ABB RobotStudio station: COMPAS_RRC_IRB-4600-40_2.55_ws_zhaw_hslu.rspag

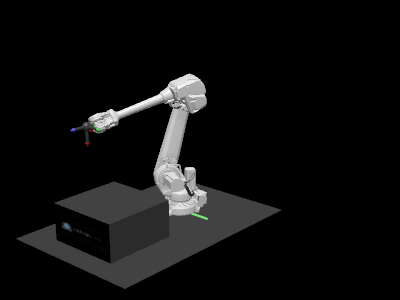
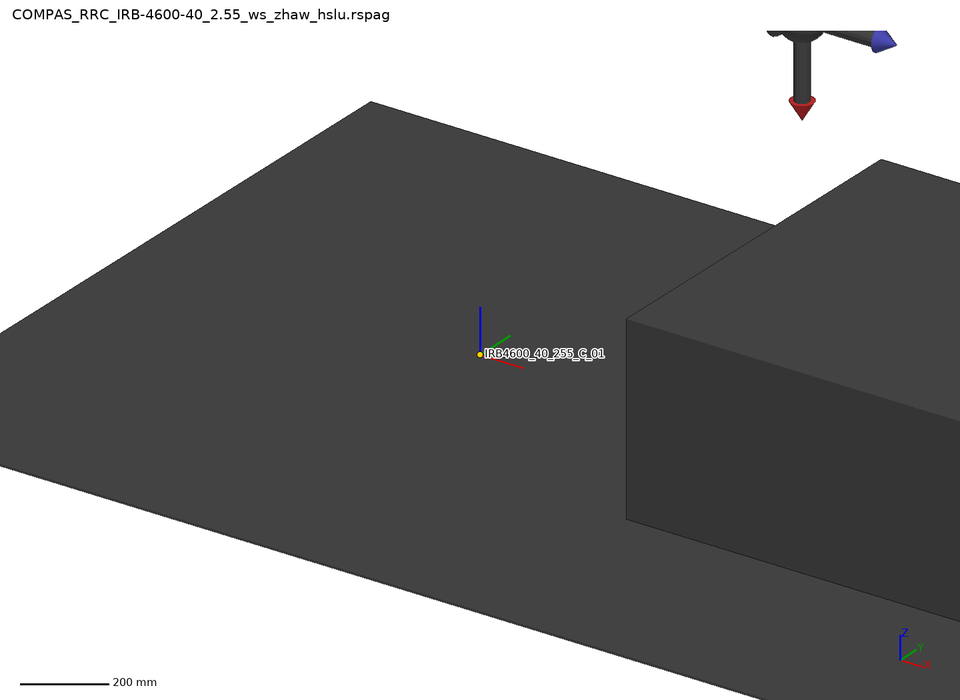
[picture v1: parts stored in the station drawn from their meshes, with robot base, taught points and paths (robot models come from the ABB library and are not in the file)]
--- station ---
Station COMPAS_RRC_IRB-4600-40_2.55 (saved by RobotStudio 22.2.10013.1)
Controller vIRB4600-40-2.55-RW11
  mechanical unit ROB_1: IRB4600_40_255_C_01, 6 joints, base frame (0, 0, 0) mm
Layout (positions relative to the parent item):
  - IRB4600_40_255_C_01 [mechanism] at (0, 0, 0) mm; joint values [-0.4275, -0.3109, 0.5805, -1.0418, -0.501, 0.9829] (rad or m)
      links: Base, Link1, Link2, Link3, Link4, Link5, Link6
  - Tool [graphiccomponentgroup] at (1145.78, -460.56, 1367.89) mm, rotated rx -105.47 ry 90 rz -105.47 deg
    - Tool X [part], size 50 x 60 x 60 mm
    - Tool Y [part], size 60 x 50 x 60 mm
    - Tool Z [part], size 60 x 60 x 50 mm
    - Base [part] at (1428.26, 0, 1185.08) mm, rotated rx 180 ry 0 rz -180 deg, size 272.5 x 272.4 x 270 mm
    - Tool X TubeTrace [smart component]
        properties: TraceObject=(none); ActiveTube=(none); Mechanism=IRB4600_40_255_C_01; Flange=Tool0; Parent=(none); Flange Offset=[0.26 0 0.06]; Tube Diameter=0.03; Color (RGB)=[255 255 255]; Color=-65536; Min Distance=0.001; Redraw Rate (ms)=10; NoOfBodies=278; Remove Geometry=true; Transient=false
        signals: DI Execute, DI NewTrace, DI Clear, DO TraceCreated
    - Tool Y TubeTrace [smart component]
        properties: TraceObject=(none); ActiveTube=(none); Mechanism=IRB4600_40_255_C_01; Flange=Tool0; Parent=(none); Flange Offset=[0 0.26 0.06]; Tube Diameter=0.03; Color (RGB)=[255 255 255]; Color=-16711872; Min Distance=0.001; Redraw Rate (ms)=10; NoOfBodies=278; Remove Geometry=true; Transient=false
        signals: DI Execute, DI NewTrace, DI Clear, DO TraceCreated
    - Tool Z TubeTrace [smart component]
        properties: TraceObject=(none); ActiveTube=(none); Mechanism=IRB4600_40_255_C_01; Flange=Tool0; Parent=(none); Flange Offset=[0 0 0.32]; Tube Diameter=0.03; Color (RGB)=[255 255 255]; Color=-16776961; Min Distance=0.001; Redraw Rate (ms)=10; NoOfBodies=278; Remove Geometry=true; Transient=false
        signals: DI Execute, DI NewTrace, DI Clear, DO TraceCreated
  - Example_Setup [graphiccomponentgroup]
    - Ground [part], size 3000 x 2000 x 5 mm
    - Table [part], size 1000 x 1000 x 500 mm
Attachment: Tool is attached to IRB4600_40_255_C_01 / Link6
Station logic (signal -> signal, property => property):
  vIRB4600-40-2.55-RW11.do_X -> Tool X TubeTrace.Execute
  vIRB4600-40-2.55-RW11.do_Y -> Tool Y TubeTrace.Execute
  vIRB4600-40-2.55-RW11.do_Z -> Tool Z TubeTrace.Execute

--- Backups/vIRB4600-40-2.55-RW11/RAPID/TASK1/PROGMOD/RRC_Example.mod ---
MODULE RRC_Example
    !***********************************************************************************
    !
    ! ETH Zurich / Robotic Fabrication Lab
    ! HIB C 13 / Stefano-Franscini-Platz 1
    ! CH-8093 Zurich
    !
    !***********************************************************************************
    !
    ! PROJECT     :  RRC - Rapid Robot Communication
    !
    ! FUNCTION    :  Example modul for the project
    !
    ! AUTHOR      :  Philippe Fleischmann
    !
    ! EMAIL       :  rrc@arch.ethz.ch
    !
    ! HISTORY     :  2019.02.22
    !
    ! Copyright   :  ETH Zurich (CH) 2019
    !                - Philippe Fleischmann
    !                - Michael Lyrenmann
    !                - Gonzalo Casas
    !
    ! License     :  This code base is governed by an EULA (End-User License Agreement)
    !                which you have received together with the software.
    !                You are not allowed to use the software on a real robots
    !                without a signed EULA.
    !
    !                A copy of the EULA content is in the controller task (T_CTRL).
    !
    !***********************************************************************************

    !************************************************
    ! Declaration :     tooldata
    !************************************************
    !
    TASK PERS tooldata t_RRC_Tool_X:=[TRUE,[[260,0,60],[0.707106781,0,0.707106781,0]],[15,[0,0,60],[1,0,0,0],0,0,0]];
    TASK PERS tooldata t_RRC_Tool_Y:=[TRUE,[[0,260,60],[0.707106781,-0.707106781,0,0]],[15,[0,0,60],[1,0,0,0],0,0,0]];
    TASK PERS tooldata t_RRC_Tool_Z:=[TRUE,[[0,0,320],[1,0,0,0]],[15,[0,0,60],[1,0,0,0],0,0,0]];

    !************************************************
    ! Declaration :     wobjdata
    !************************************************
    !
    TASK PERS wobjdata ob_RRC_Workplace:=[FALSE,TRUE,"",[[750,-500,500],[1,0,0,0]],[[0,0,0],[1,0,0,0]]];

ENDMODULE

--- Backups/vIRB4600-40-2.55-RW11/RAPID/TASK1/PROGMOD/RRC_Main.mod ---
MODULE RRC_Main
    !***********************************************************************************
    !
    ! ETH Zurich / Robotic Fabrication Lab
    ! HIB C 13 / Stefano-Franscini-Platz 1
    ! CH-8093 Zurich
    !
    !***********************************************************************************
    !
    ! PROJECT     :  RRC - Rapid Robot Communication
    !
    ! FUNCTION    :  Main modul for the project
    !
    ! AUTHOR      :  Philippe Fleischmann
    !
    ! EMAIL       :  rrc@arch.ethz.ch
    !
    ! HISTORY     :  2019.02.22
    !
    ! Copyright   :  ETH Zurich (CH) 2019
    !                - Philippe Fleischmann
    !                - Michael Lyrenmann
    !                - Gonzalo Casas
    !
    ! License     :  This code base is governed by an EULA (End-User License Agreement)
    !                which you have received together with the software.
    !                You are not allowed to use the software on a real robots
    !                without a signed EULA.
    !
    !                A copy of the EULA content is in the controller task (T_CTRL).
    !
    !***********************************************************************************

    !************************************************
    ! Function    :     main
    ! Programmer  :     Philippe Fleischmann
    ! Date        :     2019.02.22
    !***************** ETH Zurich *******************
    !
    PROC main()
        !****************************!
        !                            !
        !   #####   #####    ####    !
        !   #    #  #    #  #    #   !
        !   #    #  #    #  #        !
        !   #####   #####   #        !
        !   #   #   #   #   #    #   !
        !   #    #  #    #   ####    !
        !                            !
        !****************************!
        !
        r_RRC_Main;
    ENDPROC

ENDMODULE

--- Backups/vIRB4600-40-2.55-RW11/RAPID/TASK1/SYSMOD/RRC_Base_DataTask_Rob.sys ---
MODULE RRC_Base_DataTask_Rob (SYSMODULE)
    !***********************************************************************************
    !
    ! ETH Zurich / Robotic Fabrication Lab
    ! HIB C 13 / Stefano-Franscini-Platz 1
    ! CH-8093 Zurich
    !
    !***********************************************************************************
    !
    ! PROJECT     :  RRC - Rapid Robot Communication
    !
    ! FUNCTION    :  Base Data Task Library
    !
    ! AUTHOR      :  Philippe Fleischmann
    !
    ! EMAIL       :  rrc@arch.ethz.ch
    !
    ! HISTORY     :  2019.02.22
    !
    ! Copyright   :  ETH Zurich (CH) 2019
    !                - Philippe Fleischmann
    !                - Michael Lyrenmann
    !                - Gonzalo Casas
    !
    ! License     :  This code base is governed by an EULA (End-User License Agreement)
    !                which you have received together with the software.
    !                You are not allowed to use the software on a real robots
    !                without a signed EULA.
    !
    !                A copy of the EULA content is in the controller task (T_CTRL).
    !
    !***********************************************************************************

    !************************************************
    ! Declaration :     num
    !************************************************
    !
    TASK PERS num n_RRC_Answer:=0;
    TASK PERS num n_RRC_Act_S_ID:=4;
    TASK PERS num n_RRC_Time:=1;
    TASK PERS num n_RRC_Acc:=100;
    TASK PERS num n_RRC_Ramp:=100;
    TASK PERS num n_RRC_Override:=100;
    TASK PERS num n_RRC_MaxTCP:=500;
    TASK PERS num n_RRC_FloatValue:=42;

    !************************************************
    ! Declaration :     string
    !************************************************
    !
    TASK PERS string st_RRC_UIAnswer:="Set my Speed";
    TASK PERS string st_RRC_ActMsg1:="Requested speed is not posible, minimal value is 0.1 mm/s";
    TASK PERS string st_RRC_ActMsg2:="Submited speed : 0.0 mm/s";
    TASK PERS string st_RRC_ActMsg3:="";
    TASK PERS string st_RRC_ActMsg4:="";
    TASK PERS string st_RRC_ActMsg5:="";
    TASK PERS string st_RRC_ActBtn1:="50 mm/s";
    TASK PERS string st_RRC_ActBtn2:="100 mm/s";
    TASK PERS string st_RRC_ActBtn3:="Set my Speed";
    TASK PERS string st_RRC_ActBtn4:="";
    TASK PERS string st_RRC_ActBtn5:="";
    TASK PERS string st_RRC_Header:="Update Speed";
    TASK PERS string st_RRC_TPWrite:="Moving to position on target_frame";
    TASK PERS string st_RRC_StringValue:="Custom Text";

    !************************************************
    ! Declaration :     tooldata
    !************************************************
    !
    TASK PERS tooldata t_RRC_Act:=[TRUE,[[0,0,320],[1,0,0,0]],[15,[0,0,60],[1,0,0,0],0,0,0]];

    !************************************************
    ! Declaration :     wobjdata
    !************************************************
    !
    TASK PERS wobjdata ob_RRC_Act:=[FALSE,TRUE,"",[[750,-500,500],[1,0,0,0]],[[0,0,0],[1,0,0,0]]];

    !************************************************
    ! Declaration :     speeddata
    !************************************************
    !
    CONST speeddata v_RRC_Default:=[25,500,5000,1000];
    TASK PERS speeddata v_RRC_Act:=[200,500,5000,1000];

    !************************************************
    ! Declaration :     zonedata
    !************************************************
    !
    TASK PERS zonedata z_RRC_Act:=[TRUE,0,0,0,0,0,0];

    !************************************************
    ! Declaration :     jointtarget
    !************************************************
    !
    TASK PERS jointtarget jp_RRC_Act:=[[-24.4963,-17.8131,33.2614,-59.6898,-28.7042,56.3166],[9E+9,9E+9,9E+9,9E+9,9E+9,9E+9]];

    !************************************************
    ! Declaration :     robtarget
    !************************************************
    !
    TASK PERS robtarget p_RRC_Act:=[[715.775,39.4411,867.894],[0.707107,0,0.707107,0],[0,0,-1,0],[9E+9,9E+9,9E+9,9E+9,9E+9,9E+9]];

    !************************************************
    ! Declaration :     signaldo
    !************************************************
    !
    VAR signaldo do_RRC_Act;

    !************************************************
    ! Declaration :     signalgo
    !************************************************
    !
    VAR signalgo go_RRC_Act;

    !************************************************
    ! Declaration :     signalao
    !************************************************
    !
    VAR signalao ao_RRC_Act;

    !************************************************
    ! Declaration :     signaldi
    !************************************************
    !
    VAR signaldi di_RRC_Act;

    !************************************************
    ! Declaration :     signalgi
    !************************************************
    !
    VAR signalgi gi_RRC_Act;

    !************************************************
    ! Declaration :     signalai
    !************************************************
    !
    VAR signalai ai_RRC_Act;

    !************************************************
    ! Declaration :     signalai
    !************************************************
    !
    VAR clock ck_RRC_StopWatch;

ENDMODULE

--- Backups/vIRB4600-40-2.55-RW11/RAPID/TASK1/SYSMOD/RRC_Base_Feedback_Rob.sys ---
MODULE RRC_Base_Feedback_Rob(SYSMODULE)
    !***********************************************************************************
    !
    ! ETH Zurich / Robotic Fabrication Lab
    ! HIB C 13 / Stefano-Franscini-Platz 1
    ! CH-8093 Zurich
    !
    !***********************************************************************************
    !
    ! PROJECT     :  RRC - Rapid Robot Communication
    !
    ! FUNCTION    :  Base Feedback Library
    !
    ! AUTHOR      :  Philippe Fleischmann
    !
    ! EMAIL       :  rrc@arch.ethz.ch
    !
    ! HISTORY     :  2019.02.22
    !
    ! Copyright   :  ETH Zurich (CH) 2019
    !                - Philippe Fleischmann
    !                - Michael Lyrenmann
    !                - Gonzalo Casas
    !
    ! License     :  This code base is governed by an EULA (End-User License Agreement)
    !                which you have received together with the software.
    !                You are not allowed to use the software on a real robots
    !                without a signed EULA.
    !
    !                A copy of the EULA content is in the controller task (T_CTRL).
    !
    !***********************************************************************************

    !************************************************
    ! Function    :     Feedback add string
    ! Programmer  :     Philippe Fleischmann
    ! Date        :     2019.02.22
    !***************** ETH Zurich *******************
    !
    PROC r_RRC_FAddString(string stString)
        !
        ! Increase feedback string counter
        Incr n_RRC_CounterFStr;
        !
        ! Select string to add
        TEST n_RRC_CounterFStr
        CASE 1:
            !
            ! Add string
            bm_RRC_ActSenMsgRob.Data.St1:=stString;
        CASE 2:
            !
            ! Add string
            bm_RRC_ActSenMsgRob.Data.St2:=stString;
        CASE 3:
            !
            ! Add string
            bm_RRC_ActSenMsgRob.Data.St3:=stString;
        CASE 4:
            !
            ! Add string
            bm_RRC_ActSenMsgRob.Data.St4:=stString;
        CASE 5:
            !
            ! Add string
            bm_RRC_ActSenMsgRob.Data.St5:=stString;
        DEFAULT:
            !
            ! Program error
            r_RRC_ProgError;
        ENDTEST
        !
        ! Update string counter
        bm_RRC_ActSenMsgRob.Data.St_Cnt:=n_RRC_CounterFStr;
        RETURN ;
    ERROR
        ! Placeholder for Error Code...
    ENDPROC

    !************************************************
    ! Function    :     Feedback add value
    ! Programmer  :     Philippe Fleischmann
    ! Date        :     2019.02.22
    !***************** ETH Zurich *******************
    !
    PROC r_RRC_FAddValue(num nValue)
        !
        ! Increase feedback value counter
        Incr n_RRC_CounterFVal;
        !
        ! Select value to add
        TEST n_RRC_CounterFVal
        CASE 1:
            !
            ! Add value
            bm_RRC_ActSenMsgRob.Data.V1:=nValue;
        CASE 2:
            !
            ! Add value
            bm_RRC_ActSenMsgRob.Data.V2:=nValue;
        CASE 3:
            !
            ! Add value
            bm_RRC_ActSenMsgRob.Data.V3:=nValue;
        CASE 4:
            !
            ! Add value
            bm_RRC_ActSenMsgRob.Data.V4:=nValue;
        CASE 5:
            !
            ! Add value
            bm_RRC_ActSenMsgRob.Data.V5:=nValue;
        CASE 6:
            !
            ! Add value
            bm_RRC_ActSenMsgRob.Data.V6:=nValue;
        CASE 7:
            !
            ! Add value
            bm_RRC_ActSenMsgRob.Data.V7:=nValue;
        CASE 8:
            !
            ! Add value
            bm_RRC_ActSenMsgRob.Data.V8:=nValue;
        CASE 9:
            !
            ! Add value
            bm_RRC_ActSenMsgRob.Data.V9:=nValue;
        CASE 10:
            !
            ! Add value
            bm_RRC_ActSenMsgRob.Data.V10:=nValue;
        CASE 11:
            !
            ! Add value
            bm_RRC_ActSenMsgRob.Data.V11:=nValue;
        CASE 12:
            !
            ! Add value
            bm_RRC_ActSenMsgRob.Data.V12:=nValue;
        CASE 13:
            !
            ! Add value
            bm_RRC_ActSenMsgRob.Data.V13:=nValue;
        CASE 14:
            !
            ! Add value
            bm_RRC_ActSenMsgRob.Data.V14:=nValue;
        CASE 15:
            !
            ! Add value
            bm_RRC_ActSenMsgRob.Data.V15:=nValue;
        CASE 16:
            !
            ! Add value
            bm_RRC_ActSenMsgRob.Data.V16:=nValue;
        CASE 17:
            !
            ! Add value
            bm_RRC_ActSenMsgRob.Data.V17:=nValue;
        CASE 18:
            !
            ! Add value
            bm_RRC_ActSenMsgRob.Data.V18:=nValue;
        CASE 19:
            !
            ! Add value
            bm_RRC_ActSenMsgRob.Data.V19:=nValue;
        CASE 20:
            !
            ! Add value
            bm_RRC_ActSenMsgRob.Data.V20:=nValue;
        CASE 21:
            !
            ! Add value
            bm_RRC_ActSenMsgRob.Data.V21:=nValue;
        CASE 22:
            !
            ! Add value
            bm_RRC_ActSenMsgRob.Data.V22:=nValue;
        CASE 23:
            !
            ! Add value
            bm_RRC_ActSenMsgRob.Data.V23:=nValue;
        CASE 24:
            !
            ! Add value
            bm_RRC_ActSenMsgRob.Data.V24:=nValue;
        CASE 25:
            !
            ! Add value
            bm_RRC_ActSenMsgRob.Data.V25:=nValue;
        CASE 26:
            !
            ! Add value
            bm_RRC_ActSenMsgRob.Data.V26:=nValue;
        CASE 27:
            !
            ! Add value
            bm_RRC_ActSenMsgRob.Data.V27:=nValue;
        CASE 28:
            !
            ! Add value
            bm_RRC_ActSenMsgRob.Data.V28:=nValue;
        CASE 29:
            !
            ! Add value
            bm_RRC_ActSenMsgRob.Data.V29:=nValue;
        CASE 30:
            !
            ! Add value
            bm_RRC_ActSenMsgRob.Data.V30:=nValue;
        DEFAULT:
            !
            ! Program error
            r_RRC_ProgError;
        ENDTEST
        !
        ! Update value counter
        bm_RRC_ActSenMsgRob.Data.V_Cnt:=n_RRC_CounterFVal;
        RETURN ;
    ERROR
        ! Placeholder for Error Code...
    ENDPROC

    !************************************************
    ! Function    :     Feedback done
    ! Programmer  :     Philippe Fleischmann
    ! Date        :     2019.02.22
    !***************** ETH Zurich *******************
    !
    PROC r_RRC_FDone()
        !
        ! Add Sqz_ID from Client in Feedback ID
        bm_RRC_ActSenMsgRob.Data.F_ID:=bm_RRC_RecBufferRob{n_RRC_ChaNr,n_RRC_ReadPtrRecBuf}.Data.S_ID;
        !
        ! Instruction
        bm_RRC_ActSenMsgRob.Data.Instr:=bm_RRC_RecBufferRob{n_RRC_ChaNr,n_RRC_ReadPtrRecBuf}.Data.Instr;
        !
        ! Feedback
        bm_RRC_ActSenMsgRob.Data.Feedb:="Done";
        RETURN ;
    ERROR
        ! Placeholder for Error Code...
    ENDPROC

    !************************************************
    ! Function    :     Feedback Position
    ! Programmer  :     Philippe Fleischmann
    ! Date        :     2019.02.22
    !***************** ETH Zurich *******************
    !
    PROC r_RRC_FPos(num nFL)
        !
        ! Check feedback level
        TEST nFL
        CASE 10001:
            !
            ! add robot position after robot is in position
            r_RRC_FActRobT;
        CASE 10002:
            !
            ! add fly by robot positon
            r_RRC_FActRobT\FlyBy;
        CASE 10003:
            !
            ! add robot joints after robot is in position
            r_RRC_FActJointT;
        CASE 10004:
            !
            ! add fly by joints positon
            r_RRC_FActJointT\FlyBy;
        ENDTEST
        RETURN ;
    ERROR
        ! Placeholder for Error Code...
    ENDPROC

    !************************************************
    ! Function    :     Feedback actual jointtarget
    ! Programmer  :     Philippe Fleischmann
    ! Date        :     2019.02.22
    !***************** ETH Zurich *******************
    !
    PROC r_RRC_FActJointT(\switch FlyBy)
        !
        ! Read actual jointtartet
        r_RRC_ReadActJointT\FlyBy?FlyBy;
        !
        ! Read robot axis
        r_RRC_FAddValue jp_RRC_Act.robax.rax_1;
        r_RRC_FAddValue jp_RRC_Act.robax.rax_2;
        r_RRC_FAddValue jp_RRC_Act.robax.rax_3;
        r_RRC_FAddValue jp_RRC_Act.robax.rax_4;
        r_RRC_FAddValue jp_RRC_Act.robax.rax_5;
        r_RRC_FAddValue jp_RRC_Act.robax.rax_6;
        !
        ! Read external axis
        r_RRC_FAddValue jp_RRC_Act.extax.eax_a;
        r_RRC_FAddValue jp_RRC_Act.extax.eax_b;
        r_RRC_FAddValue jp_RRC_Act.extax.eax_c;
        !
        ! Reserve for unused external axis
        r_RRC_FAddValue jp_RRC_Act.extax.eax_d;
        r_RRC_FAddValue jp_RRC_Act.extax.eax_e;
        r_RRC_FAddValue jp_RRC_Act.extax.eax_f;
        RETURN ;
    ERROR
        ! Placeholder for Error Code...
    ENDPROC

    !************************************************
    ! Function    :     Feedback actual robtarget
    ! Programmer  :     Philippe Fleischmann
    ! Date        :     2019.02.22
    !***************** ETH Zurich *******************
    !
    PROC r_RRC_FActRobT(\switch FlyBy)
        !
        ! Read actual robtarget
        r_RRC_ReadActRobT\FlyBy?FlyBy;
        !
        ! Read actual translation
        r_RRC_FAddValue p_RRC_Act.trans.x;
        r_RRC_FAddValue p_RRC_Act.trans.y;
        r_RRC_FAddValue p_RRC_Act.trans.z;
        !
        ! Read actual rotation (Quaternions)
        r_RRC_FAddValue p_RRC_Act.rot.q1;
        r_RRC_FAddValue p_RRC_Act.rot.q2;
        r_RRC_FAddValue p_RRC_Act.rot.q3;
        r_RRC_FAddValue p_RRC_Act.rot.q4;
        !
        ! Read actual external axis
        r_RRC_FAddValue p_RRC_Act.extax.eax_a;
        r_RRC_FAddValue p_RRC_Act.extax.eax_b;
        r_RRC_FAddValue p_RRC_Act.extax.eax_c;
        !
        ! Reserve for unused external axis
        r_RRC_FAddValue p_RRC_Act.extax.eax_d;
        r_RRC_FAddValue p_RRC_Act.extax.eax_e;
        r_RRC_FAddValue p_RRC_Act.extax.eax_f;
        RETURN ;
    ERROR
        ! Placeholder for Error Code...
    ENDPROC

    !************************************************
    ! Function    :     Feedback error
    ! Programmer  :     Philippe Fleischmann
    ! Date        :     2019.02.22
    !***************** ETH Zurich *******************
    !
    PROC r_RRC_FError()
        !
        ! Feedback error with feedback code
        bm_RRC_ActSenMsgRob.Data.Feedb:="Done FError "+NumToStr(bm_RRC_RecBufferRob{n_RRC_ChaNr,n_RRC_ReadPtrRecBuf}.Data.F_Lev,0);
        RETURN ;
    ERROR
        ! Placeholder for Error Code...
    ENDPROC
ENDMODULE

--- Backups/vIRB4600-40-2.55-RW11/RAPID/TASK1/SYSMOD/RRC_Base_Instructions_Rob.sys ---
MODULE RRC_Base_Instructions_Rob(SYSMODULE)
    !***********************************************************************************
    !
    ! ETH Zurich / Robotic Fabrication Lab
    ! HIB C 13 / Stefano-Franscini-Platz 1
    ! CH-8093 Zurich
    !
    !***********************************************************************************
    !
    ! PROJECT     :  RRC - Rapid Robot Communication
    !
    ! FUNCTION    :  Base Instracion Library
    !
    ! AUTHOR      :  Philippe Fleischmann
    !
    ! EMAIL       :  rrc@arch.ethz.ch
    !
    ! HISTORY     :  2019.02.22
    !
    ! Copyright   :  ETH Zurich (CH) 2019
    !                - Philippe Fleischmann
    !                - Michael Lyrenmann
    !                - Gonzalo Casas
    !
    ! License     :  This code base is governed by an EULA (End-User License Agreement)
    !                which you have received together with the software.
    !                You are not allowed to use the software on a real robots
    !                without a signed EULA.
    !
    !                A copy of the EULA content is in the controller task (T_CTRL).
    !
    !***********************************************************************************

    !************************************************
    ! Function    :     Move to Joints (MoveAbsJ)
    ! Programmer  :     Philippe Fleischmann
    ! Date        :     2019.02.22
    !***************** ETH Zurich *******************
    !
    PROC r_RRC_MoveToJoints()
        !
        ! Read and set jonttarget
        r_RRC_RasJointtarget;
        !
        ! Read and set tcp speed
        r_RRC_RasTCPSpeed bm_RRC_RecBufferRob{n_RRC_ChaNr,n_RRC_ReadPtrRecBuf}.Data.V13;
        !
        ! Read and set zone
        r_RRC_RasZone bm_RRC_RecBufferRob{n_RRC_ChaNr,n_RRC_ReadPtrRecBuf}.Data.V14;
        !
        ! Move robot
        MoveAbsJ jp_RRC_Act,v_RRC_Act,z_RRC_Act,t_RRC_Act;
        !
        ! Feedback
        IF bm_RRC_RecBufferRob{n_RRC_ChaNr,n_RRC_ReadPtrRecBuf}.Data.F_Lev>0 THEN
            !
            ! Instruction done
            r_RRC_FDone;
            !
            ! Check additional feedback
            IF bm_RRC_RecBufferRob{n_RRC_ChaNr,n_RRC_ReadPtrRecBuf}.Data.F_Lev>1 THEN
                !
                ! Cenerate feedback
                TEST bm_RRC_RecBufferRob{n_RRC_ChaNr,n_RRC_ReadPtrRecBuf}.Data.F_Lev
                DEFAULT:
                    !
                    ! Not defined
                    !
                    ! Feedback not supported
                    r_RRC_FError;
                ENDTEST
            ENDIF
            !
            ! Move message in send buffer
            r_RRC_MovMsgToSenBufRob n_RRC_ChaNr;
        ENDIF
        RETURN ;
    ERROR
        ! Placeholder for Error Code...
    ENDPROC

    !************************************************
    ! Function    :     Move to (MoveL or MoveJ)
    ! Programmer  :     Philippe Fleischmann
    ! Date        :     2019.02.22
    !***************** ETH Zurich *******************
    !
    PROC r_RRC_MoveTo()
        !
        ! Read and set robtarget
        r_RRC_RASRobtarget\stMoveType:=bm_RRC_RecBufferRob{n_RRC_ChaNr,n_RRC_ReadPtrRecBuf}.Data.st1;
        !
        ! Read and set tcp speed
        r_RRC_RasTCPSpeed bm_RRC_RecBufferRob{n_RRC_ChaNr,n_RRC_ReadPtrRecBuf}.Data.V14;
        !
        ! Read and set zone
        r_RRC_RasZone bm_RRC_RecBufferRob{n_RRC_ChaNr,n_RRC_ReadPtrRecBuf}.Data.V15;
        !
        ! Select move type
        IF bm_RRC_RecBufferRob{n_RRC_ChaNr,n_RRC_ReadPtrRecBuf}.Data.st1="L" OR bm_RRC_RecBufferRob{n_RRC_ChaNr,n_RRC_ReadPtrRecBuf}.Data.st1="FrameL" THEN
            !
            ! Linear
            !
            !
            ! Deactivate configuration check
            ConfL\Off;
            !
            ! Move robot
            MoveL p_RRC_Act,v_RRC_Act,z_RRC_Act,t_RRC_Act\WObj:=ob_RRC_Act;
            !
            ! Activate configuration check
            ConfL\On;
        ELSE
            !
            ! Joint
            !
            !
            ! Deactivate configuration check
            ConfJ\Off;
            !
            ! Move robot
            MoveJ p_RRC_Act,v_RRC_Act,z_RRC_Act,t_RRC_Act\WObj:=ob_RRC_Act;
            !
            ! Activate configuration check
            ConfJ\On;
        ENDIF
        !
        ! Feedback
        IF bm_RRC_RecBufferRob{n_RRC_ChaNr,n_RRC_ReadPtrRecBuf}.Data.F_Lev>0 THEN
            !
            ! Instruction done
            r_RRC_FDone;
            !
            ! Check additional feedback
            IF bm_RRC_RecBufferRob{n_RRC_ChaNr,n_RRC_ReadPtrRecBuf}.Data.F_Lev>1 THEN
                !
                ! Cenerate feedback
                TEST bm_RRC_RecBufferRob{n_RRC_ChaNr,n_RRC_ReadPtrRecBuf}.Data.F_Lev
                DEFAULT:
                    !
                    ! Not defined
                    !
                    ! Feedback not supported
                    r_RRC_FError;
                ENDTEST
            ENDIF
            !
            ! Move message in send buffer
            r_RRC_MovMsgToSenBufRob n_RRC_ChaNr;
        ENDIF
        RETURN ;
    ERROR
        ! Placeholder for Error Code...
    ENDPROC

    !************************************************
    ! Function    :     Set analog output (SetAO)
    ! Programmer  :     Philippe Fleischmann
    ! Date        :     2019.02.22
    !***************** ETH Zurich *******************
    !
    PROC r_RRC_SetAnalog()
        !
        ! Get actual output
        GetDataVal bm_RRC_RecBufferRob{n_RRC_ChaNr,n_RRC_ReadPtrRecBuf}.Data.St1,ao_RRC_Act;
        !
        ! Set actual output
        SetAO ao_RRC_Act,bm_RRC_RecBufferRob{n_RRC_ChaNr,n_RRC_ReadPtrRecBuf}.Data.V1;
        !
        ! Feedback
        IF bm_RRC_RecBufferRob{n_RRC_ChaNr,n_RRC_ReadPtrRecBuf}.Data.F_Lev>0 THEN
            !
            ! Cenerate feedback
            TEST bm_RRC_RecBufferRob{n_RRC_ChaNr,n_RRC_ReadPtrRecBuf}.Data.F_Lev
            CASE 1:
                !
                ! Instruction done
                r_RRC_FDone;
            DEFAULT:
                !
                ! Feedback not supported
                r_RRC_FError;
            ENDTEST
            !
            ! Move message in send buffer
            r_RRC_MovMsgToSenBufRob n_RRC_ChaNr;
        ENDIF
        RETURN ;
    ERROR
        ! Placeholder for Error Code...
    ENDPROC

    !************************************************
    ! Function    :     Read ananlog input ((AInput)
    ! Programmer  :     Philippe Fleischmann
    ! Date        :     2019.02.22
    !***************** ETH Zurich *******************
    !
    PROC r_RRC_ReadAnalog()
        !
        ! Get actual output
        GetDataVal bm_RRC_RecBufferRob{n_RRC_ChaNr,n_RRC_ReadPtrRecBuf}.Data.St1,ai_RRC_Act;
        !
        ! Add standard feedback instruction done
        r_RRC_FDone;
        !
        ! Read input value and add it to feedback
        r_RRC_FAddValue AInput(ai_RRC_Act);
        !
        ! Feedback
        IF bm_RRC_RecBufferRob{n_RRC_ChaNr,n_RRC_ReadPtrRecBuf}.Data.F_Lev>1 THEN
            !
            ! Check additional feedback
            TEST bm_RRC_RecBufferRob{n_RRC_ChaNr,n_RRC_ReadPtrRecBuf}.Data.F_Lev
            CASE 10001,10002,10003,10004:
                !
                ! add robot position
                r_RRC_FPos bm_RRC_RecBufferRob{n_RRC_ChaNr,n_RRC_ReadPtrRecBuf}.Data.F_Lev;
            DEFAULT:
                !
                ! Not defined
                !
                ! Feedback not supported
                r_RRC_FError;
            ENDTEST
        ENDIF
        !
        ! Move message in send buffer
        r_RRC_MovMsgToSenBufRob n_RRC_ChaNr;
        RETURN ;
    ERROR
        ! Placeholder for Error Code...
    ENDPROC

    !************************************************
    ! Function    :     Set group output (SetGO)
    ! Programmer  :     Philippe Fleischmann
    ! Date        :     2019.02.22
    !***************** ETH Zurich *******************
    !
    PROC r_RRC_SetGroup()
        !
        ! Get actual output
        GetDataVal bm_RRC_RecBufferRob{n_RRC_ChaNr,n_RRC_ReadPtrRecBuf}.Data.St1,go_RRC_Act;
        !
        ! Set actual output
        SetGO go_RRC_Act,bm_RRC_RecBufferRob{n_RRC_ChaNr,n_RRC_ReadPtrRecBuf}.Data.V1;
        !
        ! Feedback
        IF bm_RRC_RecBufferRob{n_RRC_ChaNr,n_RRC_ReadPtrRecBuf}.Data.F_Lev>0 THEN
            !
            ! Cenerate feedback
            TEST bm_RRC_RecBufferRob{n_RRC_ChaNr,n_RRC_ReadPtrRecBuf}.Data.F_Lev
            CASE 1:
                !
                ! Instruction done
                r_RRC_FDone;
            DEFAULT:
                !
                ! Feedback not supported
                r_RRC_FError;
            ENDTEST
            !
            ! Move message in send buffer
            r_RRC_MovMsgToSenBufRob n_RRC_ChaNr;
        ENDIF
        RETURN ;
    ERROR
        ! Placeholder for Error Code...
    ENDPROC

    !************************************************
    ! Function    :     Read group input (GInput)
    ! Programmer  :     Philippe Fleischmann
    ! Date        :     2019.02.22
    !***************** ETH Zurich *******************
    !
    PROC r_RRC_ReadGroup()
        !
        ! Get actual output
        GetDataVal bm_RRC_RecBufferRob{n_RRC_ChaNr,n_RRC_ReadPtrRecBuf}.Data.St1,gi_RRC_Act;
        !
        ! Add standard feedback instruction done
        r_RRC_FDone;
        !
        ! Read input value and add it to feedback
        r_RRC_FAddValue GInput(gi_RRC_Act);
        !
        ! Feedback
        IF bm_RRC_RecBufferRob{n_RRC_ChaNr,n_RRC_ReadPtrRecBuf}.Data.F_Lev>1 THEN
            !
            ! Check additional feedback
            TEST bm_RRC_RecBufferRob{n_RRC_ChaNr,n_RRC_ReadPtrRecBuf}.Data.F_Lev
            CASE 10001,10002,10003,10004:
                !
                ! add robot position
                r_RRC_FPos bm_RRC_RecBufferRob{n_RRC_ChaNr,n_RRC_ReadPtrRecBuf}.Data.F_Lev;
            DEFAULT:
                !
                ! Not defined
                !
                ! Feedback not supported
                r_RRC_FError;
            ENDTEST
        ENDIF
        !
        ! Move message in send buffer
        r_RRC_MovMsgToSenBufRob n_RRC_ChaNr;
        RETURN ;
    ERROR
        ! Placeholder for Error Code...
    ENDPROC

    !************************************************
    ! Function    :     Set digital output (SetDO)
    ! Programmer  :     Philippe Fleischmann
    ! Date        :     2019.02.22
    !***************** ETH Zurich *******************
    !
    PROC r_RRC_SetDigital()
        !
        ! Get actual output
        GetDataVal bm_RRC_RecBufferRob{n_RRC_ChaNr,n_RRC_ReadPtrRecBuf}.Data.St1,do_RRC_Act;
        !
        ! Set actual output
        SetDO do_RRC_Act,bm_RRC_RecBufferRob{n_RRC_ChaNr,n_RRC_ReadPtrRecBuf}.Data.V1;
        !
        ! Feedback
        IF bm_RRC_RecBufferRob{n_RRC_ChaNr,n_RRC_ReadPtrRecBuf}.Data.F_Lev>0 THEN
            !
            ! Cenerate feedback
            TEST bm_RRC_RecBufferRob{n_RRC_ChaNr,n_RRC_ReadPtrRecBuf}.Data.F_Lev
            CASE 1:
                !
                ! Instruction done
                r_RRC_FDone;
            DEFAULT:
                !
                ! Feedback not supported
                r_RRC_FError;
            ENDTEST
            !
            ! Move message in send buffer
            r_RRC_MovMsgToSenBufRob n_RRC_ChaNr;
        ENDIF
        RETURN ;
    ERROR
        ! Placeholder for Error Code...
    ENDPROC

    !************************************************
    ! Function    :     Pulse digital output (PulsDo)
    ! Programmer  :     Philippe Fleischmann
    ! Date        :     2019.02.22
    !***************** ETH Zurich *******************
    !
    PROC r_RRC_PulseDigital()
        !
        ! Get actual output
        GetDataVal bm_RRC_RecBufferRob{n_RRC_ChaNr,n_RRC_ReadPtrRecBuf}.Data.St1,do_RRC_Act;
        !
        ! Set actual output
        PulseDO\High\PLength:=bm_RRC_RecBufferRob{n_RRC_ChaNr,n_RRC_ReadPtrRecBuf}.Data.V1,do_RRC_Act;
        !
        ! Feedback
        IF bm_RRC_RecBufferRob{n_RRC_ChaNr,n_RRC_ReadPtrRecBuf}.Data.F_Lev>0 THEN
            !
            ! Cenerate feedback
            TEST bm_RRC_RecBufferRob{n_RRC_ChaNr,n_RRC_ReadPtrRecBuf}.Data.F_Lev
            CASE 1:
                !
                ! Instruction done
                r_RRC_FDone;
            DEFAULT:
                !
                ! Feedback not supported
                r_RRC_FError;
            ENDTEST
            !
            ! Move message in send buffer
            r_RRC_MovMsgToSenBufRob n_RRC_ChaNr;
        ENDIF
        RETURN ;
    ERROR
        ! Placeholder for Error Code...
    ENDPROC

    !************************************************
    ! Function    :     Read digital input (DInput)
    ! Programmer  :     Philippe Fleischmann
    ! Date        :     2019.02.22
    !***************** ETH Zurich *******************
    !
    PROC r_RRC_ReadDigital()
        !
        ! Get actual output
        GetDataVal bm_RRC_RecBufferRob{n_RRC_ChaNr,n_RRC_ReadPtrRecBuf}.Data.St1,di_RRC_Act;
        !
        ! Add standard feedback instruction done
        r_RRC_FDone;
        !
        ! Read input value and add it to feedback
        r_RRC_FAddValue DInput(Di_RRC_Act);
        !
        ! Feedback
        IF bm_RRC_RecBufferRob{n_RRC_ChaNr,n_RRC_ReadPtrRecBuf}.Data.F_Lev>1 THEN
            !
            ! Check additional feedback
            TEST bm_RRC_RecBufferRob{n_RRC_ChaNr,n_RRC_ReadPtrRecBuf}.Data.F_Lev
            CASE 10001,10002,10003,10004:
                !
                ! add robot position
                r_RRC_FPos bm_RRC_RecBufferRob{n_RRC_ChaNr,n_RRC_ReadPtrRecBuf}.Data.F_Lev;
            DEFAULT:
                !
                ! Not defined
                ! Feedback not supported
                r_RRC_FError;
            ENDTEST
        ENDIF
        !
        ! Move message in send buffer
        r_RRC_MovMsgToSenBufRob n_RRC_ChaNr;
        RETURN ;
    ERROR
        ! Placeholder for Error Code...
    ENDPROC

    !************************************************
    ! Function    :     Set tool (tooldata)
    ! Programmer  :     Philippe Fleischmann
    ! Date        :     2019.02.22
    !***************** ETH Zurich *******************
    !
    PROC r_RRC_SetTool()
        VAR tooldata tX:=[TRUE,[[0,0,0],[1,0,0,0]],[0,[0,0,0],[1,0,0,0],0,0,0]];
        !
        ! Get tool
        GetDataVal bm_RRC_RecBufferRob{n_RRC_ChaNr,n_RRC_ReadPtrRecBuf}.Data.St1,tX;
        !
        ! Set t_RRC_Act
        t_RRC_Act:=tX;
        !
        ! Feedback
        IF bm_RRC_RecBufferRob{n_RRC_ChaNr,n_RRC_ReadPtrRecBuf}.Data.F_Lev>0 THEN
            !
            ! Instruction done
            r_RRC_FDone;
            !
            ! Check additional feedback
            IF bm_RRC_RecBufferRob{n_RRC_ChaNr,n_RRC_ReadPtrRecBuf}.Data.F_Lev>1 THEN
                !
                ! Cenerate feedback
                TEST bm_RRC_RecBufferRob{n_RRC_ChaNr,n_RRC_ReadPtrRecBuf}.Data.F_Lev
                CASE 10001:
                    !
                    ! Tooldata
                    ! String 1 from Client
                    r_RRC_FAddString bm_RRC_RecBufferRob{n_RRC_ChaNr,n_RRC_ReadPtrRecBuf}.Data.St1;
                    !
                    ! String 2 Structure of parameter information
                    r_RRC_FAddString "Feedback -Tool -Robhold -Pos -Orient -Mass";
                    !
                    ! String 3 roboter hold tool yes or no
                    IF t_RRC_Act.robhold=TRUE r_RRC_FAddString "Yes";
                    IF t_RRC_Act.robhold=FALSE r_RRC_FAddString "No";
                    !
                    ! Value 1..3 TCP position xyz
                    r_RRC_FAddValue t_RRC_Act.tframe.trans.x;
                    r_RRC_FAddValue t_RRC_Act.tframe.trans.y;
                    r_RRC_FAddValue t_RRC_Act.tframe.trans.z;
                    !
                    ! Value 4..7 TCP orientation q1..q4
                    r_RRC_FAddValue t_RRC_Act.tframe.rot.q1;
                    r_RRC_FAddValue t_RRC_Act.tframe.rot.q2;
                    r_RRC_FAddValue t_RRC_Act.tframe.rot.q3;
                    r_RRC_FAddValue t_RRC_Act.tframe.rot.q4;
                    !
                    ! Value 8 Tool mass
                    r_RRC_FAddValue t_RRC_Act.tload.mass;
                DEFAULT:
                    !
                    ! Feedback not supported
                    r_RRC_FError;
                ENDTEST
            ENDIF
            !
            ! Move message in send buffer
            r_RRC_MovMsgToSenBufRob n_RRC_ChaNr;
        ENDIF
        RETURN ;
    ERROR
        ! Placeholder for Error Code...
    ENDPROC

    !************************************************
    ! Function    :     Set work object (wobjdata)
    ! Programmer  :     Philippe Fleischmann
    ! Date        :     2019.02.22
    !***************** ETH Zurich *******************
    !
    PROC r_RRC_SetWorkObject()
        VAR wobjdata obX:=[FALSE,TRUE,"",[[0,0,0],[1,0,0,0]],[[0,0,0],[1,0,0,0]]];
        !
        ! Get workobject
        GetDataVal bm_RRC_RecBufferRob{n_RRC_ChaNr,n_RRC_ReadPtrRecBuf}.Data.St1,obX;
        !
        ! Set ob_RRC_Act
        ob_RRC_Act:=obX;
        !
        ! Feedback
        IF bm_RRC_RecBufferRob{n_RRC_ChaNr,n_RRC_ReadPtrRecBuf}.Data.F_Lev>0 THEN
            !
            ! Instruction done
            r_RRC_FDone;
            !
            ! Check additional feedback
            IF bm_RRC_RecBufferRob{n_RRC_ChaNr,n_RRC_ReadPtrRecBuf}.Data.F_Lev>1 THEN
                !
                ! Cenerate feedback
                TEST bm_RRC_RecBufferRob{n_RRC_ChaNr,n_RRC_ReadPtrRecBuf}.Data.F_Lev
                CASE 10001:
                    !
                    ! Wobjdata
                    ! String 1 from Client
                    r_RRC_FAddString bm_RRC_RecBufferRob{n_RRC_ChaNr,n_RRC_ReadPtrRecBuf}.Data.St1;
                    !
                    ! String 2 Structure of parameter information
                    r_RRC_FAddString "Feedback Workobject -Robhold -UFProg -UFMec -UFPos -UFOrient -OFPos -OFOrient";
                    !
                    ! String 3 roboter hold workobject yes or no
                    IF ob_RRC_Act.robhold=TRUE r_RRC_FAddString "Yes";
                    IF ob_RRC_Act.robhold=FALSE r_RRC_FAddString "No";
                    !
                    ! String 4 roboter user frame used yes or no
                    IF ob_RRC_Act.ufprog=TRUE r_RRC_FAddString "Yes";
                    IF ob_RRC_Act.ufprog=FALSE r_RRC_FAddString "No";
                    !
                    ! String 5 user frame mechanic
                    r_RRC_FAddString ob_RRC_Act.ufmec;
                    !
                    ! Value 1..3 user frame position xyz
                    r_RRC_FAddValue ob_RRC_Act.uframe.trans.x;
                    r_RRC_FAddValue ob_RRC_Act.uframe.trans.y;
                    r_RRC_FAddValue ob_RRC_Act.uframe.trans.z;
                    !
                    ! Value 4..7 user frame orientation q1..q4
                    r_RRC_FAddValue ob_RRC_Act.uframe.rot.q1;
                    r_RRC_FAddValue ob_RRC_Act.uframe.rot.q2;
                    r_RRC_FAddValue ob_RRC_Act.uframe.rot.q3;
                    r_RRC_FAddValue ob_RRC_Act.uframe.rot.q4;
                    !
                    ! Value 8..10 object frame position xyz
                    r_RRC_FAddValue ob_RRC_Act.oframe.trans.x;
                    r_RRC_FAddValue ob_RRC_Act.oframe.trans.y;
                    r_RRC_FAddValue ob_RRC_Act.oframe.trans.z;
                    !
                    ! Value 11..14 object frame orientation q1..q4
                    r_RRC_FAddValue ob_RRC_Act.oframe.rot.q1;
                    r_RRC_FAddValue ob_RRC_Act.oframe.rot.q2;
                    r_RRC_FAddValue ob_RRC_Act.oframe.rot.q3;
                    r_RRC_FAddValue ob_RRC_Act.oframe.rot.q4;
                DEFAULT:
                    !
                    ! Feedback not supported
                    r_RRC_FError;
                ENDTEST
            ENDIF
            !
            ! Move message in send buffer
            r_RRC_MovMsgToSenBufRob n_RRC_ChaNr;
        ENDIF
        RETURN ;
    ERROR
        ! Placeholder for Error Code...
    ENDPROC

    !************************************************
    ! Function    :     Get robtarget (CRobT)
    ! Programmer  :     Philippe Fleischmann
    ! Date        :     2019.02.22
    !***************** ETH Zurich *******************
    !
    PROC r_RRC_GetRobtarget()
        !
        ! Add standard feedback instruction done
        r_RRC_FDone;
        !
        ! Get robtarget
        IF bm_RRC_RecBufferRob{n_RRC_ChaNr,n_RRC_ReadPtrRecBuf}.Data.V1=1 THEN
            !
            ! Fly by
            r_RRC_FActRobT\FlyBy;
        ELSE
            !
            ! In positinton
            r_RRC_FActRobT;
        ENDIF
        !
        ! Feedback
        IF bm_RRC_RecBufferRob{n_RRC_ChaNr,n_RRC_ReadPtrRecBuf}.Data.F_Lev>1 THEN
            !
            ! Check additional feedback
            TEST bm_RRC_RecBufferRob{n_RRC_ChaNr,n_RRC_ReadPtrRecBuf}.Data.F_Lev
            DEFAULT:
                !
                ! Not defined
                !
                ! Feedback not supported
                r_RRC_FError;
            ENDTEST
        ENDIF
        !
        ! Move message in send buffer
        r_RRC_MovMsgToSenBufRob n_RRC_ChaNr;
        RETURN ;
    ERROR
        ! Placeholder for Error Code...
    ENDPROC

    !************************************************
    ! Function    :     Get joints (CJoinT)
    ! Programmer  :     Philippe Fleischmann
    ! Date        :     2019.02.22
    !***************** ETH Zurich *******************
    !
    PROC r_RRC_GetJoints()
        !
        ! Add standard feedback instruction done
        r_RRC_FDone;
        !
        ! Get robtarget
        IF bm_RRC_RecBufferRob{n_RRC_ChaNr,n_RRC_ReadPtrRecBuf}.Data.V1=1 THEN
            !
            ! Fly by
            r_RRC_FActJointT\FlyBy;
        ELSE
            !
            ! In positinton
            r_RRC_FActJointT;
        ENDIF
        !
        ! Feedback
        IF bm_RRC_RecBufferRob{n_RRC_ChaNr,n_RRC_ReadPtrRecBuf}.Data.F_Lev>1 THEN
            !
            ! Check additional feedback
            TEST bm_RRC_RecBufferRob{n_RRC_ChaNr,n_RRC_ReadPtrRecBuf}.Data.F_Lev
            DEFAULT:
                !
                ! Not defined
                !
                ! Feedback not supported
                r_RRC_FError;
            ENDTEST
        ENDIF
        !
        ! Move message in send buffer
        r_RRC_MovMsgToSenBufRob n_RRC_ChaNr;
        RETURN ;
    ERROR
        ! Placeholder for Error Code...
    ENDPROC

    !************************************************
    ! Function    :     Start Stopwatch (ClkStart)
    ! Programmer  :     Philippe Fleischmann
    ! Date        :     2019.02.22
    !***************** ETH Zurich *******************
    !
    PROC r_RRC_StartWatch()
        !
        ! Reset and start watch
        ClkReset ck_RRC_StopWatch;
        ClkStart ck_RRC_StopWatch;
        !
        ! Feedback
        IF bm_RRC_RecBufferRob{n_RRC_ChaNr,n_RRC_ReadPtrRecBuf}.Data.F_Lev>0 THEN
            !
            ! Add standard feedback instruction done
            r_RRC_FDone;
            !
            ! Feedback
            IF bm_RRC_RecBufferRob{n_RRC_ChaNr,n_RRC_ReadPtrRecBuf}.Data.F_Lev>1 THEN
                !
                ! Check additional feedback
                TEST bm_RRC_RecBufferRob{n_RRC_ChaNr,n_RRC_ReadPtrRecBuf}.Data.F_Lev
                CASE 10001,10002,10003,10004:
                    !
                    ! add robot position
                    r_RRC_FPos bm_RRC_RecBufferRob{n_RRC_ChaNr,n_RRC_ReadPtrRecBuf}.Data.F_Lev;
                DEFAULT:
                    !
                    ! Not defined
                    ! Feedback not supported
                    r_RRC_FError;
                ENDTEST
            ENDIF
            !
            ! Move message in send buffer
            r_RRC_MovMsgToSenBufRob n_RRC_ChaNr;
        ENDIF
        RETURN ;
    ERROR
        ! Placeholder for Error Code...
    ENDPROC

    !************************************************
    ! Function    :     Stop Stopwatch (ClkStop)
    ! Programmer  :     Philippe Fleischmann
    ! Date        :     2019.02.22
    !***************** ETH Zurich *******************
    !
    PROC r_RRC_StopWatch()
        !
        ! Stop watch and read time
        ClkStop ck_RRC_StopWatch;
        !
        ! Add standard feedback instruction done
        r_RRC_FDone;
        !
        ! Read stop wacht time and add it to feedback
        bm_RRC_ActSenMsgRob.Data.V1:=ClkRead(ck_RRC_StopWatch);
        !
        ! Feedback
        IF bm_RRC_RecBufferRob{n_RRC_ChaNr,n_RRC_ReadPtrRecBuf}.Data.F_Lev>0 THEN
            !
            ! Add standard feedback instruction done
            r_RRC_FDone;
            !
            ! Feedback
            IF bm_RRC_RecBufferRob{n_RRC_ChaNr,n_RRC_ReadPtrRecBuf}.Data.F_Lev>1 THEN
                !
                ! Check additional feedback
                TEST bm_RRC_RecBufferRob{n_RRC_ChaNr,n_RRC_ReadPtrRecBuf}.Data.F_Lev
                CASE 10001,10002,10003,10004:
                    !
                    ! add robot position
                    r_RRC_FPos bm_RRC_RecBufferRob{n_RRC_ChaNr,n_RRC_ReadPtrRecBuf}.Data.F_Lev;
                DEFAULT:
                    !
                    ! Not defined
                    ! Feedback not supported
                    r_RRC_FError;
                ENDTEST
            ENDIF
            !
            ! Move message in send buffer
            r_RRC_MovMsgToSenBufRob n_RRC_ChaNr;
        ENDIF
        RETURN ;
    ERROR
        ! Placeholder for Error Code...
    ENDPROC

    !************************************************
    ! Function    :     Read Watch (ClkRead)
    ! Programmer  :     Philippe Fleischmann
    ! Date        :     2019.02.22
    !***************** ETH Zurich *******************
    !
    PROC r_RRC_ReadWatch()
        !
        ! Read stop wacht time and add it to feedback
        r_RRC_FAddValue ClkRead(ck_RRC_StopWatch);
        !
        ! Feedback
        IF bm_RRC_RecBufferRob{n_RRC_ChaNr,n_RRC_ReadPtrRecBuf}.Data.F_Lev>0 THEN
            !
            ! Add standard feedback instruction done
            r_RRC_FDone;
            !
            ! Feedback
            IF bm_RRC_RecBufferRob{n_RRC_ChaNr,n_RRC_ReadPtrRecBuf}.Data.F_Lev>1 THEN
                !
                ! Check additional feedback
                TEST bm_RRC_RecBufferRob{n_RRC_ChaNr,n_RRC_ReadPtrRecBuf}.Data.F_Lev
                CASE 10001,10002,10003,10004:
                    !
                    ! add robot position
                    r_RRC_FPos bm_RRC_RecBufferRob{n_RRC_ChaNr,n_RRC_ReadPtrRecBuf}.Data.F_Lev;
                DEFAULT:
                    !
                    ! Not defined
                    ! Feedback not supported
                    r_RRC_FError;
                ENDTEST
            ENDIF
            !
            ! Move message in send buffer
            r_RRC_MovMsgToSenBufRob n_RRC_ChaNr;
        ENDIF
        RETURN ;
    ERROR
        ! Placeholder for Error Code...
    ENDPROC

    !************************************************
    ! Function    :     Stop (Stop)
    ! Programmer  :     Philippe Fleischmann
    ! Date        :     2019.02.22
    !***************** ETH Zurich *******************
    !
    PROC r_RRC_Stop()
        !
        ! Stop task
        Stop;
        !
        ! Feedback
        IF bm_RRC_RecBufferRob{n_RRC_ChaNr,n_RRC_ReadPtrRecBuf}.Data.F_Lev>0 THEN
            !
            ! Cenerate feedback
            TEST bm_RRC_RecBufferRob{n_RRC_ChaNr,n_RRC_ReadPtrRecBuf}.Data.F_Lev
            CASE 1:
                !
                ! Instruction done
                r_RRC_FDone;
            DEFAULT:
                !
                ! Feedback not supported
                r_RRC_FError;
            ENDTEST
            !
            ! Move message in send buffer
            r_RRC_MovMsgToSenBufRob n_RRC_ChaNr;
        ENDIF
        RETURN ;
    ERROR
        ! Placeholder for Error Code...
    ENDPROC

    !************************************************
    ! Function    :     Wait time (WaitTime)
    ! Programmer  :     Philippe Fleischmann
    ! Date        :     2019.02.22
    !***************** ETH Zurich *******************
    !
    PROC r_RRC_WaitTime()
        !
        ! Read time
        n_RRC_Time:=bm_RRC_RecBufferRob{n_RRC_ChaNr,n_RRC_ReadPtrRecBuf}.Data.V1;
        !
        ! Wait time
        WaitTime n_RRC_Time;
        !
        ! Feedback
        IF bm_RRC_RecBufferRob{n_RRC_ChaNr,n_RRC_ReadPtrRecBuf}.Data.F_Lev>0 THEN
            !
            ! Cenerate feedback
            TEST bm_RRC_RecBufferRob{n_RRC_ChaNr,n_RRC_ReadPtrRecBuf}.Data.F_Lev
            CASE 1:
                !
                ! Instruction done
                r_RRC_FDone;
            DEFAULT:
                !
                ! Feedback not supported
                r_RRC_FError;
            ENDTEST
            !
            ! Move message in send buffer
            r_RRC_MovMsgToSenBufRob n_RRC_ChaNr;
        ENDIF
        RETURN ;
    ERROR
        ! Placeholder for Error Code...
    ENDPROC

    !************************************************
    ! Function    :     Set maximal speed (VelSet)
    ! Programmer  :     Philippe Fleischmann
    ! Date        :     2019.02.22
    !***************** ETH Zurich *******************
    !
    PROC r_RRC_SetMaxSpeed()
        !
        ! Read overide
        n_RRC_Override:=bm_RRC_RecBufferRob{n_RRC_ChaNr,n_RRC_ReadPtrRecBuf}.Data.V1;
        !
        ! Read max TCP
        n_RRC_MaxTCP:=bm_RRC_RecBufferRob{n_RRC_ChaNr,n_RRC_ReadPtrRecBuf}.Data.V2;
        !
        ! Set max TCP velocity
        VelSet n_RRC_Override,n_RRC_MaxTCP;
        !
        ! Feedback
        IF bm_RRC_RecBufferRob{n_RRC_ChaNr,n_RRC_ReadPtrRecBuf}.Data.F_Lev>0 THEN
            !
            ! Cenerate feedback
            TEST bm_RRC_RecBufferRob{n_RRC_ChaNr,n_RRC_ReadPtrRecBuf}.Data.F_Lev
            CASE 1:
                !
                ! Instruction done
                r_RRC_FDone;
            DEFAULT:
                !
                ! Feedback not supported
                r_RRC_FError;
            ENDTEST
            !
            ! Move message in send buffer
            r_RRC_MovMsgToSenBufRob n_RRC_ChaNr;
        ENDIF
        RETURN ;
    ERROR
        ! Placeholder for Error Code...
    ENDPROC

    !************************************************
    ! Function    :     Set acceleration (AccSet)
    ! Programmer  :     Philippe Fleischmann
    ! Date        :     2019.02.22
    !***************** ETH Zurich *******************
    !
    PROC r_RRC_SetAcceleration()
        !
        ! Read acceleration
        n_RRC_Acc:=bm_RRC_RecBufferRob{n_RRC_ChaNr,n_RRC_ReadPtrRecBuf}.Data.V1;
        !
        ! Read acceleration ramp
        n_RRC_Ramp:=bm_RRC_RecBufferRob{n_RRC_ChaNr,n_RRC_ReadPtrRecBuf}.Data.V2;
        !
        ! Acceleration set
        AccSet n_RRC_Acc,n_RRC_Ramp;
        !
        ! Feedback
        IF bm_RRC_RecBufferRob{n_RRC_ChaNr,n_RRC_ReadPtrRecBuf}.Data.F_Lev>0 THEN
            !
            ! Cenerate feedback
            TEST bm_RRC_RecBufferRob{n_RRC_ChaNr,n_RRC_ReadPtrRecBuf}.Data.F_Lev
            CASE 1:
                !
                ! Instruction done
                r_RRC_FDone;
            DEFAULT:
                !
                ! Feedback not supported
                r_RRC_FError;
            ENDTEST
            !
            ! Move message in send buffer
            r_RRC_MovMsgToSenBufRob n_RRC_ChaNr;
        ENDIF
        RETURN ;
    ERROR
        ! Placeholder for Error Code...
    ENDPROC

    !************************************************
    ! Function    :     Print text (TPWrite)
    ! Programmer  :     Philippe Fleischmann
    ! Date        :     2019.02.22
    !***************** ETH Zurich *******************
    !
    PROC r_RRC_PrintText()
        !
        ! Read Text
        st_RRC_TPWrite:=bm_RRC_RecBufferRob{n_RRC_ChaNr,n_RRC_ReadPtrRecBuf}.Data.St1;
        !
        ! Clear panel
        TPErase;
        !
        ! Show message to user
        TPWrite st_RRC_TPWrite;
        !
        ! Feedback
        IF bm_RRC_RecBufferRob{n_RRC_ChaNr,n_RRC_ReadPtrRecBuf}.Data.F_Lev>0 THEN
            !
            ! Cenerate feedback
            TEST bm_RRC_RecBufferRob{n_RRC_ChaNr,n_RRC_ReadPtrRecBuf}.Data.F_Lev
            CASE 1:
                !
                ! Instruction done
                r_RRC_FDone;
            DEFAULT:
                !
                ! Feedback not supported
                r_RRC_FError;
            ENDTEST
            !
            ! Move message in send buffer
            r_RRC_MovMsgToSenBufRob n_RRC_ChaNr;
        ENDIF
        RETURN ;
    ERROR
        ! Placeholder for Error Code...
    ENDPROC

    !************************************************
    ! Function    :     No opteration
    ! Programmer  :     Philippe Fleischmann
    ! Date        :     2019.02.22
    !***************** ETH Zurich *******************
    !
    PROC r_RRC_Noop()
        !
        ! Just a dummy procedure for communication tests
        !
        ! Read the current Sequnce ID
        n_RRC_Act_S_ID:=bm_RRC_RecBufferRob{n_RRC_ChaNr,n_RRC_ReadPtrRecBuf}.Data.S_ID;
        !
        ! Feedback
        IF bm_RRC_RecBufferRob{n_RRC_ChaNr,n_RRC_ReadPtrRecBuf}.Data.F_Lev>0 THEN
            !
            ! Cenerate feedback
            TEST bm_RRC_RecBufferRob{n_RRC_ChaNr,n_RRC_ReadPtrRecBuf}.Data.F_Lev
            CASE 1:
                !
                ! Instruction done
                r_RRC_FDone;
            DEFAULT:
                !
                ! Feedback not supported
                r_RRC_FError;
            ENDTEST
            !
            ! Move message in send buffer
            r_RRC_MovMsgToSenBufRob n_RRC_ChaNr;
        ENDIF
        RETURN ;
    ERROR
        ! Placeholder for Error Code...
    ENDPROC

    !************************************************
    ! Function    :     Custom Instruction
    ! Programmer  :     Philippe Fleischmann
    ! Date        :     2019.02.22
    !***************** ETH Zurich *******************
    !
    PROC r_RRC_CustomInstruction()
        !
        ! Read string value
        st_RRC_StringValue:=bm_RRC_RecBufferRob{n_RRC_ChaNr,n_RRC_ReadPtrRecBuf}.Data.St1;
        !
        ! Read float value
        n_RRC_FloatValue:=bm_RRC_RecBufferRob{n_RRC_ChaNr,n_RRC_ReadPtrRecBuf}.Data.V1;
        !
        ! Placehoder for your Code
        !
        ! Feedback
        IF bm_RRC_RecBufferRob{n_RRC_ChaNr,n_RRC_ReadPtrRecBuf}.Data.F_Lev>0 THEN
            !
            ! Cenerate feedback
            TEST bm_RRC_RecBufferRob{n_RRC_ChaNr,n_RRC_ReadPtrRecBuf}.Data.F_Lev
            CASE 1:
                !
                ! Instruction done
                r_RRC_FDone;
            DEFAULT:
                !
                ! Feedback not supported
                r_RRC_FError;
            ENDTEST
            !
            ! Move message in send buffer
            r_RRC_MovMsgToSenBufRob n_RRC_ChaNr;
        ENDIF
        RETURN ;
    ERROR
        ! Placeholder for Error Code...
    ENDPROC

ENDMODULE

--- Backups/vIRB4600-40-2.55-RW11/RAPID/TASK1/SYSMOD/RRC_Base_Utilities_Rob.sys ---
MODULE RRC_Base_Utilities_Rob(SYSMODULE)
    !***********************************************************************************
    !
    ! ETH Zurich / Robotic Fabrication Lab
    ! HIB C 13 / Stefano-Franscini-Platz 1
    ! CH-8093 Zurich
    !
    !***********************************************************************************
    !
    ! PROJECT     :  RRC - Rapid Robot Communication
    !
    ! FUNCTION    :  Base Utilities Library
    !
    ! AUTHOR      :  Philippe Fleischmann
    !
    ! EMAIL       :  rrc@arch.ethz.ch
    !
    ! HISTORY     :  2019.02.22
    !
    ! Copyright   :  ETH Zurich (CH) 2019
    !                - Philippe Fleischmann
    !                - Michael Lyrenmann
    !                - Gonzalo Casas
    !
    ! License     :  This code base is governed by an EULA (End-User License Agreement)
    !                which you have received together with the software.
    !                You are not allowed to use the software on a real robots
    !                without a signed EULA.
    !
    !                A copy of the EULA content is in the controller task (T_CTRL).
    !
    !***********************************************************************************

    !************************************************
    ! Function    :     Read and set jointtarget
    ! Programmer  :     Philippe Fleischmann
    ! Date        :     2019.02.22
    !***************** ETH Zurich *******************
    !
    PROC r_RRC_RasJointtarget()
        !
        ! Read and set robot axis
        jp_RRC_Act.robax.rax_1:=bm_RRC_RecBufferRob{n_RRC_ChaNr,n_RRC_ReadPtrRecBuf}.Data.V1;
        jp_RRC_Act.robax.rax_2:=bm_RRC_RecBufferRob{n_RRC_ChaNr,n_RRC_ReadPtrRecBuf}.Data.V2;
        jp_RRC_Act.robax.rax_3:=bm_RRC_RecBufferRob{n_RRC_ChaNr,n_RRC_ReadPtrRecBuf}.Data.V3;
        jp_RRC_Act.robax.rax_4:=bm_RRC_RecBufferRob{n_RRC_ChaNr,n_RRC_ReadPtrRecBuf}.Data.V4;
        jp_RRC_Act.robax.rax_5:=bm_RRC_RecBufferRob{n_RRC_ChaNr,n_RRC_ReadPtrRecBuf}.Data.V5;
        jp_RRC_Act.robax.rax_6:=bm_RRC_RecBufferRob{n_RRC_ChaNr,n_RRC_ReadPtrRecBuf}.Data.V6;
        !
        ! Read and set external axis
        jp_RRC_Act.extax.eax_a:=bm_RRC_RecBufferRob{n_RRC_ChaNr,n_RRC_ReadPtrRecBuf}.Data.V7;
        jp_RRC_Act.extax.eax_b:=bm_RRC_RecBufferRob{n_RRC_ChaNr,n_RRC_ReadPtrRecBuf}.Data.V8;
        jp_RRC_Act.extax.eax_c:=bm_RRC_RecBufferRob{n_RRC_ChaNr,n_RRC_ReadPtrRecBuf}.Data.V9;
        jp_RRC_Act.extax.eax_d:=bm_RRC_RecBufferRob{n_RRC_ChaNr,n_RRC_ReadPtrRecBuf}.Data.V10;
        jp_RRC_Act.extax.eax_e:=bm_RRC_RecBufferRob{n_RRC_ChaNr,n_RRC_ReadPtrRecBuf}.Data.V11;
        jp_RRC_Act.extax.eax_f:=bm_RRC_RecBufferRob{n_RRC_ChaNr,n_RRC_ReadPtrRecBuf}.Data.V12;
        RETURN ;
    ERROR
        ! Placeholder for Error Code...
    ENDPROC

    !************************************************
    ! Function    :     Read and set robtarget
    ! Programmer  :     Philippe Fleischmann
    ! Date        :     2019.02.22
    !***************** ETH Zurich *******************
    !
    PROC r_RRC_RasRobtarget(\string stMoveType)
        !
        ! Read current data from receiver buffer and set translation
        p_RRC_Act.trans.x:=bm_RRC_RecBufferRob{n_RRC_ChaNr,n_RRC_ReadPtrRecBuf}.Data.V1;
        p_RRC_Act.trans.y:=bm_RRC_RecBufferRob{n_RRC_ChaNr,n_RRC_ReadPtrRecBuf}.Data.V2;
        p_RRC_Act.trans.z:=bm_RRC_RecBufferRob{n_RRC_ChaNr,n_RRC_ReadPtrRecBuf}.Data.V3;
        !
        ! Read current data from receiver buffer and set rotation (Quaternions)
        p_RRC_Act.rot.q1:=bm_RRC_RecBufferRob{n_RRC_ChaNr,n_RRC_ReadPtrRecBuf}.Data.V4;
        p_RRC_Act.rot.q2:=bm_RRC_RecBufferRob{n_RRC_ChaNr,n_RRC_ReadPtrRecBuf}.Data.V5;
        p_RRC_Act.rot.q3:=bm_RRC_RecBufferRob{n_RRC_ChaNr,n_RRC_ReadPtrRecBuf}.Data.V6;
        p_RRC_Act.rot.q4:=bm_RRC_RecBufferRob{n_RRC_ChaNr,n_RRC_ReadPtrRecBuf}.Data.V7;
        !
        ! Set externeal axis
        IF stMoveType="FrameL" OR stMoveType="FrameJ" THEN
            !
            ! Read current joints
            jp_RRC_Act:=CJointT();
            !
            ! Use current external values
            p_RRC_Act.extax:=jp_RRC_Act.extax;
        ELSE
            !
            ! Read current data from receiver buffer
            p_RRC_Act.extax.eax_a:=bm_RRC_RecBufferRob{n_RRC_ChaNr,n_RRC_ReadPtrRecBuf}.Data.V8;
            p_RRC_Act.extax.eax_b:=bm_RRC_RecBufferRob{n_RRC_ChaNr,n_RRC_ReadPtrRecBuf}.Data.V9;
            p_RRC_Act.extax.eax_c:=bm_RRC_RecBufferRob{n_RRC_ChaNr,n_RRC_ReadPtrRecBuf}.Data.V10;
            p_RRC_Act.extax.eax_d:=bm_RRC_RecBufferRob{n_RRC_ChaNr,n_RRC_ReadPtrRecBuf}.Data.V11;
            p_RRC_Act.extax.eax_e:=bm_RRC_RecBufferRob{n_RRC_ChaNr,n_RRC_ReadPtrRecBuf}.Data.V12;
            p_RRC_Act.extax.eax_f:=bm_RRC_RecBufferRob{n_RRC_ChaNr,n_RRC_ReadPtrRecBuf}.Data.V13;
        ENDIF
        RETURN ;
    ERROR
        ! Placeholder for Error Code...
    ENDPROC

    !************************************************
    ! Function    :     Update tool center point speed
    ! Programmer  :     Philippe Fleischmann
    ! Date        :     2019.02.22
    !***************** ETH Zurich *******************
    !
    PROC r_RRC_RasTCPSpeed(num nTCPSpeed)
        VAR num nSpeed;
        !
        ! Round input
        nSpeed:=Round(nTCPSpeed\Dec:=2);
        !
        ! Set speed data
        v_RRC_Act:=v_RRC_Default;
        !
        ! Sanity check
        IF nSpeed>0 THEN
            !
            ! Good set TCP speed
            v_RRC_Act.v_tcp:=nSpeed;
        ELSE
            !
            ! Not good inform user
            !
            ! Load strings for user information
            st_RRC_Header:="Update Speed";
            st_RRC_ActMsg1:="Requested speed is not posible, minimal value is 0.1 mm/s";
            st_RRC_ActMsg2:="Submited speed : "+NumToStr(nSpeed,1)+" mm/s";
            st_RRC_ActBtn1:="50 mm/s";
            st_RRC_ActBtn2:="100 mm/s";
            st_RRC_ActBtn3:="Set my Speed";
            !
            ! Show user window
            st_RRC_UIAnswer:=f_RRC_UIMsg(st_RRC_Header,st_RRC_ActMsg1\stMsgL2:=st_RRC_ActMsg2,st_RRC_ActBtn1\stBtn2:=st_RRC_ActBtn2,\stBtn3:=st_RRC_ActBtn3,iconWarning);
            !
            ! Handle user answer
            TEST st_RRC_UIAnswer
            CASE st_RRC_ActBtn1:
                !
                ! Set default value 1
                v_RRC_Act.v_tcp:=v50.v_tcp;
            CASE st_RRC_ActBtn2:
                !
                ! Set default value 2
                v_RRC_Act.v_tcp:=v100.v_tcp;
            CASE st_RRC_ActBtn3:
                !
                ! User interface to set my speed
                v_RRC_Act.v_tcp:=f_RRC_UINumEntry(st_RRC_Header,"Please enter your TCP speed.",0.1,1000,iconInfo);
            DEFAULT:
                !
                ! Program error
                r_RRC_ProgError;
            ENDTEST
        ENDIF
        RETURN ;
    ERROR
        ! Placeholder for Error Code...
    ENDPROC

    !************************************************
    ! Function    :     Read and set zone
    ! Programmer  :     Philippe Fleischmann
    ! Date        :     2019.02.22
    !***************** ETH Zurich *******************
    !
    PROC r_RRC_RasZone(num nZone)
        !
        ! Set zone data
        TEST nZone
        CASE -1:
            !
            ! Fine point
            z_RRC_Act:=fine;
        CASE 0:
            !
            ! z0
            z_RRC_Act:=z0;
        CASE 1:
            !
            ! z1
            z_RRC_Act:=z1;
        CASE 5:
            !
            ! z5
            z_RRC_Act:=z5;
        CASE 10:
            !
            ! z10
            z_RRC_Act:=z10;
        CASE 15:
            !
            ! z15
            z_RRC_Act:=z15;
        CASE 20:
            !
            ! z20
            z_RRC_Act:=z20;
        CASE 30:
            !
            ! z30
            z_RRC_Act:=z30;
        CASE 40:
            !
            ! z40
            z_RRC_Act:=z40;
        CASE 50:
            !
            ! z50
            z_RRC_Act:=z50;
        CASE 60:
            !
            ! z60
            z_RRC_Act:=z60;
        CASE 80:
            !
            ! z80
            z_RRC_Act:=z80;
        CASE 100:
            !
            ! z100
            z_RRC_Act:=z100;
        CASE 150:
            !
            ! z150
            z_RRC_Act:=z150;
        CASE 200:
            !
            ! z200
            z_RRC_Act:=z200;
        DEFAULT:
            !
            ! Use fine point as default
            z_RRC_Act:=fine;
        ENDTEST
        RETURN ;
    ERROR
        ! Placeholder for Error Code...
    ENDPROC

    !************************************************
    ! Function    :     Read actual jointtarget
    ! Programmer  :     Philippe Fleischmann
    ! Date        :     2019.02.22
    !***************** ETH Zurich *******************
    !
    PROC r_RRC_ReadActJointT(\switch FlyBy)
        !
        ! Wait for Robot in position
        IF NOT Present(FlyBy) WaitRob\InPos;
        !
        ! Read current joint position
        jp_RRC_Act:=CJointT();
        RETURN ;
    ERROR
        ! Placeholder for Error Code...
    ENDPROC

    !************************************************
    ! Function    :     Read actual robtarget
    ! Programmer  :     Philippe Fleischmann
    ! Date        :     2019.02.22
    !***************** ETH Zurich *******************
    !
    PROC r_RRC_ReadActRobT(\switch FlyBy)
        !
        ! Wait for Robot in position
        IF NOT Present(FlyBy) WaitRob\InPos;
        !
        ! Read current joint position
        p_RRC_Act:=CRobT(\Tool:=t_RRC_Act\WObj:=ob_RRC_Act);
        RETURN ;
    ERROR
        ! Placeholder for Error Code...
    ENDPROC
ENDMODULE

--- Backups/vIRB4600-40-2.55-RW11/RAPID/TASK1/SYSMOD/RRC_Control_Rob.sys ---
MODULE RRC_Control_Rob(SYSMODULE)
    !***********************************************************************************
    !
    ! ETH Zurich / Robotic Fabrication Lab
    ! HIB C 13 / Stefano-Franscini-Platz 1
    ! CH-8093 Zurich
    !
    !***********************************************************************************
    !
    ! PROJECT     :  RRC - Rapid Robot Communication
    !
    ! FUNCTION    :  Control modul for the project
    !
    ! AUTHOR      :  Philippe Fleischmann
    !
    ! EMAIL       :  rrc@arch.ethz.ch
    !
    ! HISTORY     :  2019.02.22
    !
    ! Copyright   :  ETH Zurich (CH) 2019
    !                - Philippe Fleischmann
    !                - Michael Lyrenmann
    !                - Gonzalo Casas
    !
    ! License     :  This code base is governed by an EULA (End-User License Agreement)
    !                which you have received together with the software.
    !                You are not allowed to use the software on a real robots
    !                without a signed EULA.
    !
    !                A copy of the EULA content is in the controller task (T_CTRL).
    !
    !***********************************************************************************

    !************************************************
    ! Function    :     Main for Project RRC
    ! Programmer  :     Philippe Fleischmann
    ! Date        :     2019.02.22
    !***************** ETH Zurich *******************
    !
    PROC r_RRC_Main()
        !
        ! Wait until controller has set taskliste all
        WaitTime n_RRC_TimeTaskLiAll;
        !
        ! Task synchronisation
        WaitSyncTask id_RRC_MainSta,tl_RRC_All;
        !
        ! Message for Operator
        TPWrite "RRC Main";
        !
        ! Inititalize cell
        r_RRC_InitCell;
        !
        ! Production loop
        WHILE b_RRC_Run=TRUE DO
            !
            ! Wait for job in receiver buffer
            WaitUntil bm_RRC_RecBufferRob{n_RRC_ChaNr,n_RRC_ReadPtrRecBuf}.startbit=TRUE\PollRate:=n_RRC_PulRatWaiJobRec;
            !
            ! Execute job from receiver buffer
            r_RRC_ExeJobFrmRecBuf;
        ENDWHILE
        !
        ! Message for Operator
        TPWrite "RRC End";
        !
        ! Task synchronisation
        WaitSyncTask id_RRC_MainEnd,tl_RRC_All;
        !
        RETURN ;
    ERROR
        ! Placeholder for Error Code...
    ENDPROC

    !************************************************
    ! Function    :     Initialize Cell
    ! Programmer  :     Philippe Fleischmann
    ! Date        :     2019.02.22
    !***************** ETH Zurich *******************
    !
    PROC r_RRC_InitCell()
        !
        ! Task synchronisation
        WaitSyncTask id_RRC_InitSta,tl_RRC_All;
        !
        ! Task synchronisation wait for controller data
        WaitSyncTask id_RRC_InitCtrl,tl_RRC_All;
        !
        ! Initialize Variables
        r_RRC_InitVar;
        !
        ! Connect Alias Signals from Tool
        !
        ! Task synchronisation
        WaitSyncTask id_RRC_InitEnd,tl_RRC_All;
        RETURN ;
    ERROR
        ! Placeholder for Error Code...
    ENDPROC

    !************************************************
    ! Function    :     Initialize Variables
    ! Programmer  :     Philippe Fleischmann
    ! Date        :     2019.02.22
    !***************** ETH Zurich *******************
    !
    PROC r_RRC_InitVar()
        !
        ! Reset Read pointer
        n_RRC_ReadPtrRecBuf:=1;
        !
        ! Reset Counter Feedback Value
        n_RRC_CounterFStr:=0;
        !
        ! Reset Counter Feedback Value
        n_RRC_CounterFVal:=0;
        !
        ! Clear actual sending message
        bm_RRC_ActSenMsgRob:=bm_RRC_Empty;
        !
        ! Read Taskname
        st_RRC_Taskname:=GetTaskName();
        !
        ! Update event log message header
        st_RRC_EvLogMsgHeader:="RRC -- "+st_RRC_Taskname;
        !
        ! Set channel number
        TEST st_RRC_Taskname
        CASE ch_RRC_Channels.Ch_1.T_Name:
            !
            ! Set channel nuber to task
            n_RRC_ChaNr:=ch_RRC_Channels.Ch_1.Ch_Nr;
            !
        CASE ch_RRC_Channels.Ch_2.T_Name:
            !
            ! Set channel nuber to task
            n_RRC_ChaNr:=ch_RRC_Channels.Ch_2.Ch_Nr;
            !
        CASE ch_RRC_Channels.Ch_3.T_Name:
            !
            ! Set channel nuber to task
            n_RRC_ChaNr:=ch_RRC_Channels.Ch_3.Ch_Nr;
            !
        CASE ch_RRC_Channels.Ch_4.T_Name:
            !
            ! Set channel nuber to task
            n_RRC_ChaNr:=ch_RRC_Channels.Ch_4.Ch_Nr;
            !
        DEFAULT:
            !
            ! Programm error
            r_RRC_ProgError;
        ENDTEST
        RETURN ;
    ERROR
        ! Placeholder for Error Code...
    ENDPROC

    !************************************************
    ! Function    :     Activate a job for the controller
    ! Programmer  :     Philippe Fleischmann
    ! Date        :     2019.02.22
    !***************** ETH Zurich *******************
    !
    PROC r_RRC_JobForCtrl(string stJob)
        !
        ! Reserve controller
        WaitTestAndSet b_RRC_CtrlInUse;
        !
        ! Send job to controller
        st_RRC_JobForCtrl:=stJob;
        !
        ! Start jop for controller
        b_RRC_CtrlWaitForJob:=FALSE;
        !
        ! Wait until controller is finish with job
        WaitUntil b_RRC_CtrlWaitForJob=TRUE;
        !
        ! Release controller
        b_RRC_CtrlInUse:=FALSE;
        !
        RETURN ;
    ERROR
        ! Placeholder for Error Code...
    ENDPROC

    !************************************************
    ! Function    :     Execute job from reveicer buffer
    ! Programmer  :     Philippe Fleischmann
    ! Date        :     2019.02.22
    !***************** ETH Zurich *******************
    !
    PROC r_RRC_ExeJobFrmRecBuf()
        !
        ! Call instruction
        %bm_RRC_RecBufferRob{n_RRC_ChaNr,n_RRC_ReadPtrRecBuf}.Data.Instr %;
        !
        ! Set job done
        bm_RRC_RecBufferRob{n_RRC_ChaNr,n_RRC_ReadPtrRecBuf}.startbit:=FALSE;
        !
        ! Count read pointer
        IF n_RRC_ReadPtrRecBuf<DIM(bm_RRC_RecBufferRob,2) THEN
            !
            ! Increas write pointer form buffer
            Incr n_RRC_ReadPtrRecBuf;
        ELSE
            !
            ! Restart with one
            n_RRC_ReadPtrRecBuf:=1;
        ENDIF
        RETURN ;
    ERROR
        ! Placeholder for Error Code...
    ENDPROC

    !************************************************
    ! Function    :     Move message to send buffer roboter 1
    ! Programmer  :     Philippe Fleischmann
    ! Date        :     2019.02.22
    !***************** ETH Zurich *******************
    !
    PROC r_RRC_MovMsgToSenBufRob(num nChaNr)
        !
        ! Count buffer pointer
        IF n_RRC_WritePtrSenBufRob{nChaNr}<DIM(bm_RRC_SenBufferRob,2) THEN
            !
            ! Increas write pointer form buffer
            Incr n_RRC_WritePtrSenBufRob{nChaNr};
        ELSE
            !
            ! Restart with one
            n_RRC_WritePtrSenBufRob{nChaNr}:=1;
        ENDIF
        !
        ! Check for bufferline free to write
        IF NOT bm_RRC_SenBufferRob{nChaNr,n_RRC_WritePtrSenBufRob{nChaNr}}.startbit=FALSE THEN
            !
            ! Wait for bufferline free to write
            WaitUntil bm_RRC_SenBufferRob{nChaNr,n_RRC_WritePtrSenBufRob{nChaNr}}.startbit=FALSE\PollRate:=0.004\Visualize\Header:="RRC MovMsgToSenBufRob1"\Message:="Buffer full"\Icon:=iconInfo;
        ENDIF
        !
        ! Write data in buffer
        bm_RRC_SenBufferRob{nChaNr,n_RRC_WritePtrSenBufRob{nChaNr}}.Data:=bm_RRC_ActSenMsgRob.Data;
        !
        ! Set Startbit
        bm_RRC_SenBufferRob{nChaNr,n_RRC_WritePtrSenBufRob{nChaNr}}.startbit:=TRUE;
        !
        ! Clear actual sending message
        bm_RRC_ActSenMsgRob:=bm_RRC_Empty;
        !
        ! Reset Counter Feedback String and Value
        n_RRC_CounterFStr:=0;
        n_RRC_CounterFVal:=0;
        RETURN ;
    ERROR
        ! Placeholder for Error Code...
    ENDPROC

    !************************************************
    ! Function    :     ProgError
    ! Programmer  :     Philippe Fleischmann
    ! Date        :     2019.02.22
    !***************** ETH Zurich *******************
    !
    PROC r_RRC_ProgError()
        !
        ! User Info
        TPWrite "Program Error";
        !
        ! Stop Program
        Stop;
        RETURN ;
    ERROR
        ! Placeholder for Error Code...
    ENDPROC

ENDMODULE

--- Backups/vIRB4600-40-2.55-RW11/RAPID/TASK1/SYSMOD/RRC_DataGlobal.sys ---
MODULE RRC_DataGlobal(SYSMODULE)
    !***********************************************************************************
    !
    ! ETH Zurich / Robotic Fabrication Lab
    ! HIB C13 / Stefano-Franscini-Platz 1
    ! CH-8093 Zurich
    !
    !***********************************************************************************
    !
    ! PROJECT     :  RRC - Rapid Robot Communication
    !
    ! FUNCTION    :  Inclouds all project spezific global datas
    !
    ! AUTHOR      :  Philippe Fleischmann
    !
    ! EMAIL       :  rrc@arch.ethz.ch
    !
    ! HISTORY     :  2019.02.22
    !
    ! Copyright   :  ETH Zurich (CH) 2019
    !                - Philippe Fleischmann
    !                - Michael Lyrenmann
    !                - Gonzalo Casas
    !
    ! License     :  This code base is governed by an EULA (End-User License Agreement)
    !                which you have received together with the software.
    !                You are not allowed to use the software on a real robots
    !                without a signed EULA.
    !
    !                A copy of the EULA content is in the controller task (T_CTRL).
    !
    !***********************************************************************************

    !************************************************
    ! Declaration :     bool
    !************************************************
    !
    PERS bool b_RRC_TaskReceiverOn;
    PERS bool b_RRC_TaskSenderOn;
    !
    PERS bool b_RRC_CtrlWaitForJob;
    PERS bool b_RRC_CtrlHamModOn;
    PERS bool b_RRC_CtrlInUse;
    PERS bool b_RRC_AutoIPAddress;
    PERS bool b_RRC_VirtualCustomPorts;
    !
    ! Channels
    PERS bool b_RRC_Com{n_RRC_NumOfCha};
    PERS bool b_RRC_SIDCheck{n_RRC_NumOfCha};
    PERS bool b_RRC_SIDErrorStop{n_RRC_NumOfCha};
    PERS bool b_RRC_LogPro{n_RRC_NumOfCha};
    !
    ! Client information
    PERS bool b_RRC_PPMain;
    !
    ! Activate or deactivate a event log message
    PERS bool b_RRC_EvLogReadAndUnpackTime;
    PERS bool b_RRC_EvLogPackAndSendTime;
    PERS bool b_RRC_EvLogMsgInUntilMsgOutTime;
    !
    ! Temporary to measure the feedback loop
    PERS bool b_RRC_FeedbackOut;

    !************************************************
    ! Declaration :     num
    !************************************************
    !
    PERS num n_RRC_WritePtrSenBufCtrl{n_RRC_NumOfCha};
    PERS num n_RRC_WritePtrSenBufRob{n_RRC_NumOfCha};
    PERS num n_RRC_SIDMax;
    !
    PERS num n_RRC_R1_ChaNr;
    PERS num n_RRC_R2_ChaNr;
    PERS num n_RRC_R3_ChaNr;
    PERS num n_RRC_R4_ChaNr;
    !
    PERS num n_RRC_SocketPortRec{n_RRC_NumOfCha};
    PERS num n_RRC_SocketPortSen{n_RRC_NumOfCha};
    !
    PERS num n_RRC_TimeTaskLiAll;
    PERS num n_RRC_TimeTPMsg;
    !
    PERS num n_RRC_ProtocolVersion;

    !************************************************
    ! Declaration :     string
    !************************************************
    !
    PERS string n_RRC_Version;
    !
    PERS string st_RRC_CurCtrlJob;
    PERS string st_RRC_JobForCtrl;
    !
    PERS string st_RRC_IP_Address;
    PERS string st_RRC_IP_AddressVC;
    PERS string st_RRC_IP_AddressMan;
    !
    ! System data
    PERS string st_RRC_SerialNr;
    PERS string st_RRC_SoftwareVersion;
    PERS string st_RRC_RobotWare;
    PERS string st_RRC_ControllerID;
    PERS string st_RRC_WAN_IP;
    PERS string st_RRC_ControllerLang;
    PERS string st_RRC_SystemName;

    !************************************************
    ! Declaration :     tasklist
    !************************************************
    !
    !PERS tasks tl_RRC_All{5};
    PERS tasks tl_RRC_All{7};

    !************************************************
    ! Declaration :     syncident
    !************************************************
    !
    VAR syncident id_RRC_MainSta;
    VAR syncident id_RRC_MainEnd;
    !
    VAR syncident id_RRC_InitSta;
    VAR syncident id_RRC_InitCtrl;
    VAR syncident id_RRC_InitEnd;

    !************************************************
    ! Declaration :     RRC_channel
    !************************************************
    !
    PERS RRC_channel ch_RRC_Channels;

    !************************************************
    ! Declaration :     buffer_msg
    !************************************************
    !
    ! Receiver buffer for controller
    PERS RRC_buffer_msg bm_RRC_RecBufferCtrl{n_RRC_NumOfCha,10};
    !
    ! Receiver buffer for robots
    PERS RRC_buffer_msg bm_RRC_RecBufferRob{n_RRC_NumOfCha,10};
    !
    ! Sender buffer for controller
    PERS RRC_buffer_msg bm_RRC_SenBufferCtrl{n_RRC_NumOfCha,10};
    !
    ! Sender buffer for robots
    PERS RRC_buffer_msg bm_RRC_SenBufferRob{n_RRC_NumOfCha,10};

ENDMODULE

--- Backups/vIRB4600-40-2.55-RW11/RAPID/TASK1/SYSMOD/RRC_DataRecord.sys ---
MODULE RRC_DataRecord(SYSMODULE)
    !***********************************************************************************
    !
    ! ETH Zurich / Robotic Fabrication Lab
    ! HIB C 13 / Stefano-Franscini-Platz 1
    ! CH-8093 Zurich
    !
    !***********************************************************************************
    !
    ! PROJECT     :  RRC - Rapid Robot Communication
    !
    ! FUNCTION    :  Includ all data records
    !
    ! AUTHOR      :  Philippe Fleischmann
    !
    ! EMAIL       :  rrc@arch.ethz.ch
    !
    ! HISTORY     :  2019.02.22
    !
    ! Copyright   :  ETH Zurich (CH) 2019
    !                - Philippe Fleischmann
    !                - Michael Lyrenmann
    !                - Gonzalo Casas
    !
    ! License     :  This code base is governed by an EULA (End-User License Agreement)
    !                which you have received together with the software.
    !                You are not allowed to use the software on a real robots
    !                without a signed EULA.
    !
    !                A copy of the EULA content is in the controller task (T_CTRL).
    !
    !***********************************************************************************

    !************************************************
    ! Function    :     Record RRC Channel
    ! Programmer  :     Philippe Fleischmann
    ! Date        :     2019.02.22
    !***************** ETH Zurich *******************
    !
    RECORD rrc_channel
        RRC_channeldata Ch_1;
        RRC_channeldata Ch_2;
        RRC_channeldata Ch_3;
        RRC_channeldata Ch_4;
    ENDRECORD

    !************************************************
    ! Function    :     Record RRC Channeldata
    ! Programmer  :     Philippe Fleischmann
    ! Date        :     2019.02.22
    !***************** ETH Zurich *******************
    !
    RECORD rrc_channeldata
        string T_Name;
        num Ch_Nr;
    ENDRECORD

    !************************************************
    ! Function    :     Record RRC Protocol
    ! Programmer  :     Philippe Fleischmann
    ! Date        :     2019.02.22
    !***************** ETH Zurich *******************
    !
    RECORD rrc_protocol
        rrc_header ProtocolHeader;
        rrc_data ProtocolData;
    ENDRECORD

    !************************************************
    ! Function    :     Record RRC Protocol Header
    ! Programmer  :     Philippe Fleischmann
    ! Date        :     2019.02.22
    !***************** ETH Zurich *******************
    !
    RECORD rrc_header
        num M_Len;
        num Ver;
        num TS_Sec;
        num TS_NSec;
    ENDRECORD

    !************************************************
    ! Function    :     Record RRC Protocol Data
    ! Programmer  :     Philippe Fleischmann
    ! Date        :     2019.02.22
    !***************** ETH Zurich *******************
    !
    RECORD rrc_data
        num S_ID;
        num E_Lev;
        num I_Len;
        string Instr;
        num F_Lev;
        num F_Len;
        string Feedb;
        num F_ID;
        num St_Cnt;
        num St1_Len;
        string St1;
        num St2_Len;
        string St2;
        num St3_Len;
        string St3;
        num St4_Len;
        string St4;
        num St5_Len;
        string St5;
        num St6_Len;
        string St6;
        num St7_Len;
        string St7;
        num St8_Len;
        string St8;
        num V_Cnt;
        num V1;
        num V2;
        num V3;
        num V4;
        num V5;
        num V6;
        num V7;
        num V8;
        num V9;
        num V10;
        num V11;
        num V12;
        num V13;
        num V14;
        num V15;
        num V16;
        num V17;
        num V18;
        num V19;
        num V20;
        num V21;
        num V22;
        num V23;
        num V24;
        num V25;
        num V26;
        num V27;
        num V28;
        num V29;
        num V30;
        num V31;
        num V32;
        num V33;
        num V34;
        num V35;
        num V36;
    ENDRECORD

    !************************************************
    ! Function    :     Record RRC Buffer Message
    ! Programmer  :     Philippe Fleischmann
    ! Date        :     2019.02.22
    !***************** ETH Zurich *******************
    !
    RECORD rrc_buffer_msg
        rrc_data Data;
        bool StartBit;
    ENDRECORD
ENDMODULE

--- Backups/vIRB4600-40-2.55-RW11/RAPID/TASK1/SYSMOD/RRC_DataTask_Rob.sys ---
MODULE RRC_DataTask_Rob(SYSMODULE)
    !***********************************************************************************
    !
    ! ETH Zurich / Robotic Fabrication Lab
    ! HIB C 13 / Stefano-Franscini-Platz 1
    ! CH-8093 Zurich
    !
    !***********************************************************************************
    !
    ! PROJECT     :  RRC - Rapid Robot Communication
    !
    ! FUNCTION    :  Includ all Task specific Data's
    !
    ! AUTHOR      :  Philippe Fleischmann
    !
    ! EMAIL       :  rrc@arch.ethz.ch
    !
    ! HISTORY     :  2019.02.22
    !
    ! Copyright   :  ETH Zurich (CH) 2019
    !                - Philippe Fleischmann
    !                - Michael Lyrenmann
    !                - Gonzalo Casas
    !
    ! License     :  This code base is governed by an EULA (End-User License Agreement)
    !                which you have received together with the software.
    !                You are not allowed to use the software on a real robots
    !                without a signed EULA.
    !
    !                A copy of the EULA content is in the controller task (T_CTRL).
    !
    !***********************************************************************************

    !************************************************
    ! Declaration :     bool
    !************************************************
    !
    CONST bool b_RRC_Run:=TRUE;

    !************************************************
    ! Declaration :     num
    !************************************************
    !
    CONST num n_RRC_PulRatWaiJobRec:=0.01;
    !
    TASK PERS num n_RRC_ReadPtrRecBuf:=8;
    !
    CONST num n_RRC_NumOfCha:=4;
    TASK PERS num n_RRC_ChaNr:=1;
    !
    TASK PERS num n_RRC_AccRamp:=33;
    !
    TASK PERS num n_RRC_CounterFStr:=0;
    TASK PERS num n_RRC_CounterFVal:=0;

    !************************************************
    ! Declaration :     string
    !************************************************
    !
    TASK PERS string st_RRC_Taskname:="T_ROB1";
    TASK PERS string st_RRC_EvLogMsgHeader:="RRC -- T_ROB1";

    !************************************************
    ! Declaration :     RRC_buffer_msg
    !************************************************
    !
    CONST RRC_buffer_msg bm_RRC_Empty:=[[0,0,0,"",0,0,"",0,0,0,"",0,"",0,"",0,"",0,"",0,"",0,"",0,"",0,0,0,0,0,0,0,0,0,0,0,0,0,0,0,0,0,0,0,0,0,0,0,0,0,0,0,0,0,0,0,0,0,0,0,0,0],FALSE];
    !
    TASK PERS RRC_buffer_msg bm_RRC_ActSenMsgRob:=[[0,0,0,"",0,0,"",0,0,0,"",0,"",0,"",0,"",0,"",0,"",0,"",0,"",0,0,0,0,0,0,0,0,0,0,0,0,0,0,0,0,0,0,0,0,0,0,0,0,0,0,0,0,0,0,0,0,0,0,0,0,0],FALSE];



ENDMODULE

--- Backups/vIRB4600-40-2.55-RW11/RAPID/TASK1/SYSMOD/RRC_Helper_Rob.sys ---
MODULE RRC_Helper_Rob(SYSMODULE)
    !***********************************************************************************
    !
    ! ETH Zurich / Robotic Fabrication Lab
    ! HIB C 13 / Stefano-Franscini-Platz 1
    ! CH-8093 Zurich
    !
    !***********************************************************************************
    !
    ! PROJECT     :  RRC - Rapid Robot Communication
    !
    ! FUNCTION    :  Helper routines for project
    !
    ! AUTHOR      :  Philippe Fleischmann
    !
    ! EMAIL       :  rrc@arch.ethz.ch
    !
    ! HISTORY     :  2019.02.22
    !
    ! Copyright   :  ETH Zurich (CH) 2019
    !                - Philippe Fleischmann
    !                - Michael Lyrenmann
    !                - Gonzalo Casas
    !
    ! License     :  This code base is governed by an EULA (End-User License Agreement)
    !                which you have received together with the software.
    !                You are not allowed to use the software on a real robots
    !                without a signed EULA.
    !
    !                A copy of the EULA content is in the controller task (T_CTRL).
    !
    !***********************************************************************************

    !************************************************
    ! Declaration :     num
    !************************************************
    !
    TASK PERS bool b_RRC_StoJoToArryOn:=FALSE;

    !************************************************
    ! Declaration :     num
    !************************************************
    !
    TASK PERS num n_RRC_ArryPointer:=1;

    !************************************************
    ! Declaration :     jointtarget
    !************************************************
    !
    TASK PERS jointtarget jp_RRC_Arry{51}:=[
    [[-178.155,71.7205,-139.164,9.42305E-06,-22.554,223.157],[9080,-7750,-4400,0,0,0]],
    [[-176.821,72.2054,-141.287,0.000284081,-20.9164,221.819],[9080,-7750,-4400,0,0,0]],
    [[-175.414,72.6147,-143.268,9.42305E-06,-19.3465,220.411],[9080,-7750,-4400,0,0,0]],
    [[-173.945,72.9576,-145.109,0.000284081,-17.8461,218.944],[9080,-7750,-4400,0,0,0]],
    [[-172.414,73.2404,-146.822,-8.21297E-05,-16.4157,217.415],[9080,-7750,-4400,0,0,0]],
    [[-170.819,73.4679,-148.416,-8.21297E-05,-15.0513,215.818],[9080,-7750,-4400,0,0,0]],
    [[-169.155,73.6488,-149.895,9.42305E-06,-13.7544,214.156],[9080,-7750,-4400,0,0,0]],
    [[-167.425,73.7877,-151.265,-0.000173682,-12.5213,212.424],[9080,-7750,-4400,0,0,0]],
    [[-165.624,73.8886,-152.529,9.42305E-06,-11.3601,210.624],[9080,-7750,-4400,0,0,0]],
    [[-163.754,73.958,-153.688,-0.000173682,-10.2651,208.753],[9080,-7750,-4400,0,0,0]],
    [[-161.818,73.9993,-154.757,-8.21297E-05,-9.24482,206.817],[9080,-7750,-4400,0,0,0]],
    [[-159.809,74.0186,-155.724,0.000284081,-8.29295,204.807],[9080,-7750,-4400,0,0,0]],
    [[-157.734,74.0187,-156.598,9.42305E-06,-7.41683,202.733],[9080,-7750,-4400,0,0,0]],
    [[-155.594,74.0147,-157.382,-8.21297E-05,-6.62078,200.593],[9080,-7750,-4400,0,0,0]],
    [[-153.395,73.9815,-158.081,9.42305E-06,-5.90161,198.392],[9080,-7750,-4400,0,0,0]],
    [[-151.135,73.9494,-158.686,-8.21297E-05,-5.26356,196.134],[9080,-7750,-4400,0,0,0]],
    [[-148.823,73.9148,-159.205,0.000192529,-4.70732,193.82],[9080,-7750,-4400,0,0,0]],
    [[-146.463,73.8817,-159.642,-8.21297E-05,-4.23989,191.461],[9080,-7750,-4400,0,0,0]],
    [[-144.065,73.8513,-159.989,9.42305E-06,-3.86011,189.064],[9080,-7750,-4400,0,0,0]],
    [[-141.635,73.8254,-160.258,9.42305E-06,-3.56802,186.629],[9080,-7750,-4400,0,0,0]],
    [[-139.179,73.807,-160.44,9.42305E-06,-3.36782,184.176],[9080,-7750,-4400,0,0,0]],
    [[-136.709,73.7969,-160.539,9.42305E-06,-3.26041,181.706],[9080,-7750,-4400,0,0,0]],
    [[-134.231,73.7952,-160.552,-8.21297E-05,-3.24472,179.229],[9080,-7750,-4400,0,0,0]],
    [[-131.756,73.7966,-160.486,9.42305E-06,-3.31469,176.757],[9080,-7750,-4400,0,0,0]],
    [[-129.295,73.8124,-160.339,9.42305E-06,-3.4827,174.292],[9080,-7750,-4400,0,0,0]],
    [[-126.855,73.8415,-160.099,9.42305E-06,-3.73907,171.854],[9080,-7750,-4400,0,0,0]],
    [[-124.444,73.8694,-159.781,-8.21297E-05,-4.08831,169.442],[9080,-7750,-4400,0,0,0]],
    [[-122.07,73.9026,-159.383,-0.000173682,-4.52278,167.065],[9080,-7750,-4400,0,0,0]],
    [[-119.741,73.938,-158.893,-8.21297E-05,-5.04365,164.738],[9080,-7750,-4400,0,0,0]],
    [[-117.459,73.9686,-158.316,9.42305E-06,-5.65058,162.459],[9080,-7750,-4400,0,0,0]],
    [[-115.235,73.996,-157.659,0.000192529,-6.33955,160.235],[9080,-7750,-4400,0,0,0]],
    [[-113.074,74.0154,-156.909,-0.000173682,-7.1065,158.072],[9080,-7750,-4400,0,0,0]],
    [[-110.973,74.0196,-156.066,-8.21297E-05,-7.95378,155.975],[9080,-7750,-4400,0,0,0]],
    [[-108.94,74.0172,-155.133,9.42305E-06,-8.87596,153.939],[9080,-7750,-4400,0,0,0]],
    [[-106.974,73.979,-154.107,9.42305E-06,-9.86981,151.974],[9080,-7750,-4400,0,0,0]],
    [[-105.079,73.9176,-152.98,9.42305E-06,-10.9358,150.08],[9080,-7750,-4400,0,0,0]],
    [[-103.253,73.8294,-151.76,-8.21297E-05,-12.0724,148.25],[9080,-7750,-4400,0,0,0]],
    [[-101.494,73.7055,-150.431,9.42305E-06,-13.2785,146.495],[9080,-7750,-4400,0,0,0]],
    [[-99.809,73.5413,-148.995,-8.21297E-05,-14.5482,144.806],[9080,-7750,-4400,0,0,0]],
    [[-98.187,73.3321,-147.446,-8.21297E-05,-15.8872,143.184],[9080,-7750,-4400,0,0,0]],
    [[-96.6332,73.0712,-145.78,9.42305E-06,-17.2929,141.633],[9080,-7750,-4400,0,0,0]],
    [[-95.142,72.7516,-143.987,-8.21297E-05,-18.7659,140.141],[9080,-7750,-4400,0,0,0]],
    [[-93.7151,72.3684,-142.062,-8.21297E-05,-20.3089,138.71],[9080,-7750,-4400,0,0,0]],
    [[-92.3445,71.9108,-139.99,0.000192529,-21.9221,137.343],[9080,-7750,-4400,0,0,0]],
    [[-91.0364,71.3757,-137.768,-8.21297E-05,-23.6143,136.033],[9080,-7750,-4400,0,0,0]],
    [[-89.7751,70.7454,-135.359,0.000192529,-25.3872,134.776],[9080,-7750,-4400,0,0,0]],
    [[-88.5757,70.0112,-132.764,-8.21297E-05,-27.2514,133.572],[9080,-7750,-4400,0,0,0]],
    [[-87.4216,69.1557,-129.941,9.42305E-06,-29.2191,132.421],[9080,-7750,-4400,0,0,0]],
    [[-86.3194,68.1587,-126.859,-8.21297E-05,-31.3022,131.317],[9080,-7750,-4400,0,0,0]],
    [[-85.2617,66.984,-123.457,9.42305E-06,-33.5293,130.261],[9080,-7750,-4400,0,0,0]],
    [[-84.242,65.5863,-119.643,9.42305E-06,-35.946,129.244],[9080,-7750,-4400,0,0,0]]
    ];

    !************************************************
    ! Function    :     Store jointtarget in array
    ! Programmer  :     Philippe Fleischmann
    ! Date        :     2019.02.22
    !***************** ETH Zurich *******************
    !
    PROC r_RRC_StoJoPosInArry()
        !
        ! Made always a fine point
        WaitRob\InPos;
        !
        ! Increase arry pointer
        Incr n_RRC_ArryPointer;
        !
        ! Read current position
        jp_RRC_Arry{n_RRC_ArryPointer}:=CJointT();
        ! Placehoder for Code
        RETURN ;
    ERROR
        ! Placeholder for Error Code...
    ENDPROC

    !************************************************
    ! Function    :     Store jointtarget in array
    ! Programmer  :     Philippe Fleischmann
    ! Date        :     2019.02.22
    !***************** ETH Zurich *******************
    !
    PROC r_RRC_ExeJoPosFromArry()
        !
        n_RRC_ArryPointer:=1;
        !
        WHILE n_RRC_ArryPointer<=51 DO
            MoveAbsJ jp_RRC_Arry{n_RRC_ArryPointer},vmax,z200,tool0;
            ! Increase arry pointer
            Incr n_RRC_ArryPointer;
        ENDWHILE
        !
        RETURN ;
    ERROR
        ! Placeholder for Error Code...
    ENDPROC

ENDMODULE

--- Backups/vIRB4600-40-2.55-RW11/RAPID/TASK1/SYSMOD/RRC_UserInteraction_Rob.sys ---
MODULE RRC_UserInteraction_Rob(SYSMODULE,NOSTEPIN)
    !***********************************************************************************
    !
    ! ETH Zurich / Robotic Fabrication Lab
    ! HIB C 13 / Stefano-Franscini-Platz 1
    ! CH-8093 Zurich
    !
    !***********************************************************************************
    !
    ! PROJECT     :  RRC - Rapid Robot Communication
    !
    ! FUNCTION    :  General Utilities Library
    !
    ! AUTHOR      :  Philippe Fleischmann
    !
    ! EMAIL       :  rrc@arch.ethz.ch
    !
    ! HISTORY     :  2019.02.22
    !
    ! Copyright   :  ETH Zurich (CH) 2019
    !                - Philippe Fleischmann
    !                - Michael Lyrenmann
    !                - Gonzalo Casas
    !
    ! License     :  This code base is governed by an EULA (End-User License Agreement)
    !                which you have received together with the software.
    !                You are not allowed to use the software on a real robots
    !                without a signed EULA.
    !
    !                A copy of the EULA content is in the controller task (T_CTRL).
    !
    !***********************************************************************************

    !************************************************
    ! Function    :     Teach Pendant (old FelxPendant) Message
    ! Programmer  :     Philippe Fleischmann
    ! Date        :     2019.02.22
    !***************** ETH Zurich *******************
    !
    PROC r_RRC_TPMsg(string stMsg)
        !
        ! Clear Msg Panel
        TPErase;
        !
        ! Msg for user
        TPWrite stMsg;
        !
        ! Time to read the Msg
        WaitTime n_RRC_TimeTPMsg;
        RETURN ;
    ERROR
        ! Placeholder for Error Code...
    ENDPROC

    !************************************************
    ! Function    :     Teach Pendant (old FelxPendant) Error Message
    ! Programmer  :     Philippe Fleischmann
    ! Date        :     2019.02.22
    !***************** ETH Zurich *******************
    !
    PROC r_RRC_TPErrMsg(num nErrno\switch StopTask\switch StopAllTasks)
        !
        ! Clear Msg Panel
        TPErase;
        !
        ! Write error number
        TPWrite "ERRNO = "\Num:=nErrno;
        !
        ! Stop task
        IF Present(StopTask) Stop;
        !
        ! Stop all normal tasks
        IF Present(StopAllTasks) Stop\AllMoveTasks;
        RETURN ;
    ERROR
        ! Placeholder for Error Code...
    ENDPROC

    !************************************************
    ! Function    :     Event Log Message
    ! Programmer  :     Philippe Fleischmann
    ! Date        :     2019.02.22
    !***************** ETH Zurich *******************
    !
    PROC r_RRC_EvLogMsg(string stHeader,string stMsg)
        !
        ! Msg for user
        ErrWrite\I,stHeader+" "+stMsg,"rLogMsg";
        RETURN ;
    ERROR
        ! Placeholder for Error Code...
    ENDPROC

